IF (bEnable) THEN
	IF (bNull) THEN
		F_BACnet_MultiStatePV := E_BACnet_MultistateVal.eNull;
	ELSE
		F_BACnet_MultiStatePV := MAX(nState, E_BACnet_MultistateVal.eMin);
	END_IF
ELSE
	F_BACnet_MultiStatePV := E_BACnet_MultistateVal.eNothing;
END_IF

END_FUNCTION

// POUs/Helper/NC/F_BACnet_DeviceRecipient
// Returns an initialized recipient structure.
FUNCTION F_BACnet_DeviceRecipient : ST_BACnet_Recipient
VAR_INPUT
	nDeviceInstance		: UDINT			:= BACnet_Globals.nBACnetInstId_Auto;
END_VAR

F_BACnet_DeviceRecipient.eRecipientChoice := E_BACnet_RecipientChoice.eDevice;
F_BACnet_DeviceRecipient.stEntry.nDeviceInstance := F_BACnet_GetObjId(E_BACnetObjType.ObjDevice,nDeviceInstance);

END_FUNCTION

// POUs/Helper/NC/F_BACnet_EthernetRecipient
// Returns an initialized recipient structure.
FUNCTION F_BACnet_EthernetRecipient : ST_BACnet_Recipient
VAR_INPUT
	nIPAddress1		: BYTE;
	nIPAddress2		: BYTE;
	nIPAddress3		: BYTE;
	nIPAddress4		: BYTE;
	nPort			: UINT;
	nNetworkNr		: UINT;
END_VAR
VAR
	_nPort			: POINTER TO ARRAY[0 .. 1] OF BYTE := ADR(nPort);
END_VAR

F_BACnet_EthernetRecipient.eRecipientChoice := E_BACnet_RecipientChoice.eAddress;
F_BACnet_EthernetRecipient.stEntry.stNetAddr.eChoice := E_BACnet_AddressChoice.eEthernet;
F_BACnet_EthernetRecipient.stEntry.stNetAddr.nNetworkNr := nNetworkNr;
F_BACnet_EthernetRecipient.stEntry.stNetAddr.aAddress[0] := nIPAddress1;
F_BACnet_EthernetRecipient.stEntry.stNetAddr.aAddress[1] := nIPAddress2;
F_BACnet_EthernetRecipient.stEntry.stNetAddr.aAddress[2] := nIPAddress3;
F_BACnet_EthernetRecipient.stEntry.stNetAddr.aAddress[3] := nIPAddress4;

// Swap Port-Bytes:
F_BACnet_EthernetRecipient.stEntry.stNetAddr.aAddress[4] := _nPort^[1];
F_BACnet_EthernetRecipient.stEntry.stNetAddr.aAddress[5] := _nPort^[0];

END_FUNCTION

// POUs/Helper/NC/F_BACnet_EthernetRecipientEx
// Returns an initialized recipient structure.
FUNCTION F_BACnet_EthernetRecipientEx : ST_BACnet_Recipient
VAR_INPUT
	tIPAddress		: T_IPv4AddrArr;
	nPort			: UINT;
	nNetworkNr		: UINT;
END_VAR

F_BACnet_EthernetRecipientEx := F_BACnet_EthernetRecipient(tIPAddress[0], tIPAddress[1], tIPAddress[2], tIPAddress[3], nPort, nNetworkNr);

END_FUNCTION

// POUs/Helper/Real/F_BACnet_EnRealPV
FUNCTION F_BACnet_EnRealPV : DWORD
VAR_INPUT
	bEnable	: BOOL;
	fValue	: REAL;
END_VAR
VAR
	pDword : POINTER TO DWORD;
END_VAR

IF (bEnable) THEN
	pDword := ADR(fValue);
	F_BACnet_EnRealPV := pDword^;
ELSE
	F_BACnet_EnRealPV := F_BACnet_RealNull();
END_IF

END_FUNCTION

// POUs/Helper/Real/F_BACnet_IsFinite
FUNCTION F_BACnet_IsFinite : BOOL
VAR_INPUT
	fValue		: REAL;
END_VAR
VAR
	fArg		: T_Arg;
END_VAR

fArg.cbLen := SIZEOF(fValue);
fArg.eType := ARGTYPE_REAL;
fArg.pData := ADR(fValue);
F_BACnet_IsFinite := IsFinite(fArg);

END_FUNCTION

// POUs/Helper/Real/F_BACnet_RealEQ
FUNCTION F_BACnet_RealEQ : BOOL
VAR_INPUT
	fIn1	: REAL;
	fIn2	: REAL;
END_VAR
VAR
END_VAR

IF (F_BACnet_IsFinite(fIn1) <> F_BACnet_IsFinite(fIn2)) THEN
	F_BACnet_RealEQ := FALSE;
	RETURN;
END_IF
IF F_BACnet_IsFinite(fIn1) THEN
	IF (fIn1 <> fIn2) THEN
		F_BACnet_RealEQ := FALSE;
		RETURN;
	END_IF
END_IF
F_BACnet_RealEQ := TRUE;

END_FUNCTION

// POUs/Helper/Real/F_BACnet_RealGE
FUNCTION F_BACnet_RealGE : BOOL
VAR_INPUT
	fIn1	: REAL;
	fIn2	: REAL;
END_VAR
VAR
END_VAR

IF NOT (F_BACnet_IsFinite(fIn1) OR F_BACnet_IsFinite(fIn2)) THEN
	F_BACnet_RealGE := FALSE;
	RETURN;
END_IF
F_BACnet_RealGE := (fIn1 >= fIn2);

END_FUNCTION

// POUs/Helper/Real/F_BACnet_RealGT
FUNCTION F_BACnet_RealGT : BOOL
VAR_INPUT
	fIn1	: REAL;
	fIn2	: REAL;
END_VAR
VAR
END_VAR

IF NOT (F_BACnet_IsFinite(fIn1) OR F_BACnet_IsFinite(fIn2)) THEN
	F_BACnet_RealGT := FALSE;
	RETURN;
END_IF
F_BACnet_RealGT := (fIn1 > fIn2);

END_FUNCTION

// POUs/Helper/Real/F_BACnet_RealLE
FUNCTION F_BACnet_RealLE : BOOL
VAR_INPUT
	fIn1	: REAL;
	fIn2	: REAL;
END_VAR
VAR
END_VAR

IF NOT (F_BACnet_IsFinite(fIn1) OR F_BACnet_IsFinite(fIn2)) THEN
	F_BACnet_RealLE := FALSE;
	RETURN;
END_IF
F_BACnet_RealLE := (fIn1 <= fIn2);

END_FUNCTION

// POUs/Helper/Real/F_BACnet_RealLT
FUNCTION F_BACnet_RealLT : BOOL
VAR_INPUT
	fIn1	: REAL;
	fIn2	: REAL;
END_VAR
VAR
END_VAR

IF NOT (F_BACnet_IsFinite(fIn1) OR F_BACnet_IsFinite(fIn2)) THEN
	F_BACnet_RealLT := FALSE;
	RETURN;
END_IF
F_BACnet_RealLT := (fIn1 < fIn2);

END_FUNCTION

// POUs/Helper/Real/F_BACnet_RealNothing
FUNCTION F_BACnet_RealNothing : DWORD

F_BACnet_RealNothing:=16#7FFFFFFF;

END_FUNCTION

// POUs/Helper/Real/F_BACnet_RealPV
FUNCTION F_BACnet_RealPV : DWORD
VAR_INPUT
	bEnable	: BOOL; (* TRUE = commit to stack, FALSE = do-nothing *)
	bNull	: BOOL; (* TRUE = clear priority, FALSE = write value from input *)
	fValue	: REAL;
END_VAR
VAR
	pDword : POINTER TO DWORD;
END_VAR

IF (bEnable) THEN
	IF (bNull) THEN
		F_BACnet_RealPV := F_BACnet_RealNull();
	ELSE
		pDword := ADR(fValue);
		F_BACnet_RealPV := pDword^;
	END_IF
ELSE
	F_BACnet_RealPV := F_BACnet_RealNothing();
END_IF

END_FUNCTION

// POUs/Helper/Real/F_BACnet_RealToStr
FUNCTION F_BACnet_RealToStr : STRING
VAR_INPUT
	pValue	: POINTER TO REAL;
END_VAR
VAR
	fArg	: T_Arg;
	pDWORD	: POINTER TO DWORD;
END_VAR

IF (pValue <> 0) THEN
	fArg.cbLen := 4;
	fArg.eType := ARGTYPE_REAL;
	fArg.pData := pValue;
	pDWORD := pValue;
	IF IsFinite(fArg) THEN
		F_BACnet_RealToStr := REAL_TO_STRING(pValue^);
	ELSE
		IF (pDWORD^ = 16#7FFF0000) THEN
			F_BACnet_RealToStr := '#NULL';
		ELSIF (pDWORD^ AND 16#80000000) = 16#80000000 THEN
			F_BACnet_RealToStr := '-#QNAN';
		ELSE
			F_BACnet_RealToStr := '#QNAN';
		END_IF
	END_IF
END_IF

END_FUNCTION

// POUs/Helper/References/F_BACnet_Reference
FUNCTION F_BACnet_Reference : ST_BACnet_ObjectPropertyReference
VAR_INPUT
	iObject				: I_BACnet_Object;
	ePropertyId			: E_BACnetPropIdentifier		:= E_BACnetPropIdentifier.PropPresentValue;
END_VAR

F_BACnet_Reference.iObject := iObject;
F_BACnet_Reference.tObjectID := BACnet_Globals.nBACnetObjId_None;
F_BACnet_Reference.ePropertyId := ePropertyId;

END_FUNCTION

// POUs/Helper/References/F_BACnet_ReferenceByID
FUNCTION F_BACnet_ReferenceByID : ST_BACnet_ObjectPropertyReference
VAR_INPUT
	tObjectID			: T_BACnet_ObjectIdentifier;
	ePropertyId			: E_BACnetPropIdentifier		:= E_BACnetPropIdentifier.PropPresentValue;
END_VAR

F_BACnet_ReferenceByID.iObject := 0;
F_BACnet_ReferenceByID.tObjectID := tObjectID;
F_BACnet_ReferenceByID.ePropertyId := ePropertyId;

END_FUNCTION

// POUs/Helper/Scheduler/Calendar/F_BACnet_SchedCalendar
// Returns an initialized analog weekly scheduler.
FUNCTION F_BACnet_SchedCalendar : T_BACnet_SchedCalendar
VAR_INPUT
	iRefCalendar1	: I_BACnet_Cal	:= 0;
	iRefCalendar2	: I_BACnet_Cal	:= 0;
	iRefCalendar3	: I_BACnet_Cal	:= 0;
END_VAR
VAR
	nIndex			: INT;
END_VAR

F_BACnet_SchedCalendar[1].iRefCalendar := iRefCalendar1;

nIndex := 2;
IF (BACnet_Param.nSched_CalendarCount >= nIndex) THEN
	F_BACnet_SchedCalendar[nIndex].iRefCalendar := iRefCalendar2;
END_IF

nIndex := 3;
IF (BACnet_Param.nSched_CalendarCount >= nIndex) THEN
	F_BACnet_SchedCalendar[nIndex].iRefCalendar := iRefCalendar3;
END_IF

END_FUNCTION

// POUs/Helper/Scheduler/Exception/F_BACnet_SchedEntry1xA
// Returns an initialized analog weekly scheduler.
FUNCTION F_BACnet_SchedEntry1xA : T_BACnet_SchedExceptionEntryList
VAR_INPUT
	tEntry1Time		: TIME;
	fEntry1Value	: REAL;
END_VAR

F_BA_SetSchedulerEntry(F_BACnet_SchedEntry1xA[1], tEntry1Time, F_BA_RVal(fEntry1Value));

END_FUNCTION

// POUs/Helper/Scheduler/Exception/F_BACnet_SchedEntry1xB
// Returns an initialized binary weekly scheduler.
FUNCTION F_BACnet_SchedEntry1xB : T_BACnet_SchedExceptionEntryList
VAR_INPUT
	tEntry1Time		: TIME;
	bEntry1Value	: BOOL;
END_VAR

F_BA_SetSchedulerEntry(F_BACnet_SchedEntry1xB[1], tEntry1Time, F_BA_BVal(bEntry1Value));

END_FUNCTION

// POUs/Helper/Scheduler/Exception/F_BACnet_SchedEntry1xM
// Returns an initialized multistate weekly scheduler.
FUNCTION F_BACnet_SchedEntry1xM : T_BACnet_SchedExceptionEntryList
VAR_INPUT
	tEntry1Time		: TIME;
	nEntry1Value	: UDINT;
END_VAR

F_BA_SetSchedulerEntry(F_BACnet_SchedEntry1xM[1], tEntry1Time, F_BA_UDIVal(nEntry1Value));

END_FUNCTION

// POUs/Helper/Scheduler/Exception/F_BACnet_SchedEntry3xA
// Returns an initialized analog weekly scheduler.
FUNCTION F_BACnet_SchedEntry3xA : T_BACnet_SchedExceptionEntryList
VAR_INPUT
	tEntry1Time		: TIME;
	fEntry1Value	: REAL;
	tEntry2Time		: TIME;
	fEntry2Value	: REAL;
	tEntry3Time		: TIME;
	fEntry3Value	: REAL;
END_VAR

F_BA_SetSchedulerEntry(F_BACnet_SchedEntry3xA[1], tEntry1Time, F_BA_RVal(fEntry1Value));
F_BA_SetSchedulerEntry(F_BACnet_SchedEntry3xA[2], tEntry2Time, F_BA_RVal(fEntry2Value));
F_BA_SetSchedulerEntry(F_BACnet_SchedEntry3xA[3], tEntry3Time, F_BA_RVal(fEntry3Value));

END_FUNCTION

// POUs/Helper/Scheduler/Exception/F_BACnet_SchedEntry3xB
// Returns an initialized binary weekly scheduler.
FUNCTION F_BACnet_SchedEntry3xB : T_BACnet_SchedExceptionEntryList
VAR_INPUT
	tEntry1Time		: TIME;
	bEntry1Value	: BOOL;
	tEntry2Time		: TIME;
	bEntry2Value	: BOOL;
	tEntry3Time		: TIME;
	bEntry3Value	: BOOL;
END_VAR

F_BA_SetSchedulerEntry(F_BACnet_SchedEntry3xB[1], tEntry1Time, F_BA_BVal(bEntry1Value));
F_BA_SetSchedulerEntry(F_BACnet_SchedEntry3xB[2], tEntry2Time, F_BA_BVal(bEntry2Value));
F_BA_SetSchedulerEntry(F_BACnet_SchedEntry3xB[3], tEntry3Time, F_BA_BVal(bEntry3Value));

END_FUNCTION

// POUs/Helper/Scheduler/Exception/F_BACnet_SchedEntry3xM
// Returns an initialized multistate weekly scheduler.
FUNCTION F_BACnet_SchedEntry3xM : T_BACnet_SchedExceptionEntryList
VAR_INPUT
	tEntry1Time		: TIME;
	nEntry1Value	: UDINT;
	tEntry2Time		: TIME;
	nEntry2Value	: UDINT;
	tEntry3Time		: TIME;
	nEntry3Value	: UDINT;
END_VAR

F_BA_SetSchedulerEntry(F_BACnet_SchedEntry3xM[1], tEntry1Time, F_BA_UDIVal(nEntry1Value));
F_BA_SetSchedulerEntry(F_BACnet_SchedEntry3xM[2], tEntry2Time, F_BA_UDIVal(nEntry2Value));
F_BA_SetSchedulerEntry(F_BACnet_SchedEntry3xM[3], tEntry3Time, F_BA_UDIVal(nEntry3Value));

END_FUNCTION

// POUs/Helper/Scheduler/Exception/F_BACnet_SchedEntry5xA
// Returns an initialized analog weekly scheduler.
FUNCTION F_BACnet_SchedEntry5xA : T_BACnet_SchedExceptionEntryList
VAR_INPUT
	tEntry1Time		: TIME;
	fEntry1Value	: REAL;
	tEntry2Time		: TIME;
	fEntry2Value	: REAL;
	tEntry3Time		: TIME;
	fEntry3Value	: REAL;
	tEntry4Time		: TIME;
	fEntry4Value	: REAL;
	tEntry5Time		: TIME;
	fEntry5Value	: REAL;
END_VAR

F_BA_SetSchedulerEntry(F_BACnet_SchedEntry5xA[1], tEntry1Time, F_BA_RVal(fEntry1Value));
F_BA_SetSchedulerEntry(F_BACnet_SchedEntry5xA[2], tEntry2Time, F_BA_RVal(fEntry2Value));
F_BA_SetSchedulerEntry(F_BACnet_SchedEntry5xA[3], tEntry3Time, F_BA_RVal(fEntry3Value));
F_BA_SetSchedulerEntry(F_BACnet_SchedEntry5xA[4], tEntry4Time, F_BA_RVal(fEntry4Value));
F_BA_SetSchedulerEntry(F_BACnet_SchedEntry5xA[5], tEntry5Time, F_BA_RVal(fEntry5Value));

END_FUNCTION

// POUs/Helper/Scheduler/Exception/F_BACnet_SchedEntry5xB
// Returns an initialized binary weekly scheduler.
FUNCTION F_BACnet_SchedEntry5xB : T_BACnet_SchedExceptionEntryList
VAR_INPUT
	tEntry1Time		: TIME;
	bEntry1Value	: BOOL;
	tEntry2Time		: TIME;
	bEntry2Value	: BOOL;
	tEntry3Time		: TIME;
	bEntry3Value	: BOOL;
	tEntry4Time		: TIME;
	bEntry4Value	: BOOL;
	tEntry5Time		: TIME;
	bEntry5Value	: BOOL;
END_VAR

F_BA_SetSchedulerEntry(F_BACnet_SchedEntry5xB[1], tEntry1Time, F_BA_BVal(bEntry1Value));
F_BA_SetSchedulerEntry(F_BACnet_SchedEntry5xB[2], tEntry2Time, F_BA_BVal(bEntry2Value));
F_BA_SetSchedulerEntry(F_BACnet_SchedEntry5xB[3], tEntry3Time, F_BA_BVal(bEntry3Value));
F_BA_SetSchedulerEntry(F_BACnet_SchedEntry5xB[4], tEntry4Time, F_BA_BVal(bEntry4Value));
F_BA_SetSchedulerEntry(F_BACnet_SchedEntry5xB[5], tEntry5Time, F_BA_BVal(bEntry5Value));

END_FUNCTION

// POUs/Helper/Scheduler/Exception/F_BACnet_SchedEntry5xM
// Returns an initialized multistate weekly scheduler.
FUNCTION F_BACnet_SchedEntry5xM : T_BACnet_SchedExceptionEntryList
VAR_INPUT
	tEntry1Time		: TIME;
	nEntry1Value	: UDINT;
	tEntry2Time		: TIME;
	nEntry2Value	: UDINT;
	tEntry3Time		: TIME;
	nEntry3Value	: UDINT;
	tEntry4Time		: TIME;
	nEntry4Value	: UDINT;
	tEntry5Time		: TIME;
	nEntry5Value	: UDINT;
END_VAR

F_BA_SetSchedulerEntry(F_BACnet_SchedEntry5xM[1], tEntry1Time, F_BA_UDIVal(nEntry1Value));
F_BA_SetSchedulerEntry(F_BACnet_SchedEntry5xM[2], tEntry2Time, F_BA_UDIVal(nEntry2Value));
F_BA_SetSchedulerEntry(F_BACnet_SchedEntry5xM[3], tEntry3Time, F_BA_UDIVal(nEntry3Value));
F_BA_SetSchedulerEntry(F_BACnet_SchedEntry5xM[4], tEntry4Time, F_BA_UDIVal(nEntry4Value));
F_BA_SetSchedulerEntry(F_BACnet_SchedEntry5xM[5], tEntry5Time, F_BA_UDIVal(nEntry5Value));

END_FUNCTION

// POUs/Helper/Scheduler/Weekly/F_BACnet_SchedWeekly3xA
// Returns an initialized analog weekly scheduler.
FUNCTION F_BACnet_SchedWeekly3xA : T_BACnet_SchedWeek
VAR_INPUT
	eDayFrom		: E_BA_Weekday		:= E_BA_Weekday.eMonday;
	eDayTo			: E_BA_Weekday		:= E_BA_Weekday.eSunday;
	
	tEntry1Time		: TIME;
	fEntry1Value	: REAL;
	tEntry2Time		: TIME;
	fEntry2Value	: REAL;
	tEntry3Time		: TIME;
	fEntry3Value	: REAL;
END_VAR

F_BA_SetWeekdays(F_BACnet_SchedWeekly3xA, eDayFrom, eDayTo, 1, tEntry1Time, F_BA_RVal(fEntry1Value));
F_BA_SetWeekdays(F_BACnet_SchedWeekly3xA, eDayFrom, eDayTo, 2, tEntry2Time, F_BA_RVal(fEntry2Value));
F_BA_SetWeekdays(F_BACnet_SchedWeekly3xA, eDayFrom, eDayTo, 3, tEntry3Time, F_BA_RVal(fEntry3Value));

END_FUNCTION

// POUs/Helper/Scheduler/Weekly/F_BACnet_SchedWeekly3xB
// Returns an initialized binary weekly scheduler.
FUNCTION F_BACnet_SchedWeekly3xB : T_BACnet_SchedWeek
VAR_INPUT
	eDayFrom		: E_BA_Weekday		:= E_BA_Weekday.eMonday;
	eDayTo			: E_BA_Weekday		:= E_BA_Weekday.eSunday;
	
	tEntry1Time		: TIME;
	bEntry1Value	: BOOL;
	tEntry2Time		: TIME;
	bEntry2Value	: BOOL;
	tEntry3Time		: TIME;
	bEntry3Value	: BOOL;
END_VAR

F_BA_SetWeekdays(F_BACnet_SchedWeekly3xB, eDayFrom, eDayTo, 1, tEntry1Time, F_BA_BVal(bEntry1Value));
F_BA_SetWeekdays(F_BACnet_SchedWeekly3xB, eDayFrom, eDayTo, 2, tEntry2Time, F_BA_BVal(bEntry2Value));
F_BA_SetWeekdays(F_BACnet_SchedWeekly3xB, eDayFrom, eDayTo, 3, tEntry3Time, F_BA_BVal(bEntry3Value));

END_FUNCTION

// POUs/Helper/Scheduler/Weekly/F_BACnet_SchedWeekly3xM
// Returns an initialized multistate weekly scheduler.
FUNCTION F_BACnet_SchedWeekly3xM : T_BACnet_SchedWeek
VAR_INPUT
	eDayFrom		: E_BA_Weekday		:= E_BA_Weekday.eMonday;
	eDayTo			: E_BA_Weekday		:= E_BA_Weekday.eSunday;
	
	tEntry1Time		: TIME;
	nEntry1Value	: UDINT;
	tEntry2Time		: TIME;
	nEntry2Value	: UDINT;
	tEntry3Time		: TIME;
	nEntry3Value	: UDINT;
END_VAR

F_BA_SetWeekdays(F_BACnet_SchedWeekly3xM, eDayFrom, eDayTo, 1, tEntry1Time, F_BA_UDIVal(nEntry1Value));
F_BA_SetWeekdays(F_BACnet_SchedWeekly3xM, eDayFrom, eDayTo, 2, tEntry2Time, F_BA_UDIVal(nEntry2Value));
F_BA_SetWeekdays(F_BACnet_SchedWeekly3xM, eDayFrom, eDayTo, 3, tEntry3Time, F_BA_UDIVal(nEntry3Value));

END_FUNCTION

// POUs/Helper/Scheduler/Weekly/F_BACnet_SchedWeekly5xA
// Returns an initialized analog weekly scheduler.
FUNCTION F_BACnet_SchedWeekly5xA : T_BACnet_SchedWeek
VAR_INPUT
	eDayFrom		: E_BA_Weekday		:= E_BA_Weekday.eMonday;
	eDayTo			: E_BA_Weekday		:= E_BA_Weekday.eSunday;
	
	tEntry1Time		: TIME;
	fEntry1Value	: REAL;
	tEntry2Time		: TIME;
	fEntry2Value	: REAL;
	tEntry3Time		: TIME;
	fEntry3Value	: REAL;
	tEntry4Time		: TIME;
	fEntry4Value	: REAL;
	tEntry5Time		: TIME;
	fEntry5Value	: REAL;
END_VAR

F_BA_SetWeekdays(F_BACnet_SchedWeekly5xA, eDayFrom, eDayTo, 1, tEntry1Time, F_BA_RVal(fEntry1Value));
F_BA_SetWeekdays(F_BACnet_SchedWeekly5xA, eDayFrom, eDayTo, 2, tEntry2Time, F_BA_RVal(fEntry2Value));
F_BA_SetWeekdays(F_BACnet_SchedWeekly5xA, eDayFrom, eDayTo, 3, tEntry3Time, F_BA_RVal(fEntry3Value));
F_BA_SetWeekdays(F_BACnet_SchedWeekly5xA, eDayFrom, eDayTo, 4, tEntry4Time, F_BA_RVal(fEntry4Value));
F_BA_SetWeekdays(F_BACnet_SchedWeekly5xA, eDayFrom, eDayTo, 5, tEntry5Time, F_BA_RVal(fEntry5Value));

END_FUNCTION

// POUs/Helper/Scheduler/Weekly/F_BACnet_SchedWeekly5xB
// Returns an initialized binary weekly scheduler.
FUNCTION F_BACnet_SchedWeekly5xB : T_BACnet_SchedWeek
VAR_INPUT
	eDayFrom		: E_BA_Weekday		:= E_BA_Weekday.eMonday;
	eDayTo			: E_BA_Weekday		:= E_BA_Weekday.eSunday;
	
	tEntry1Time		: TIME;
	bEntry1Value	: BOOL;
	tEntry2Time		: TIME;
	bEntry2Value	: BOOL;
	tEntry3Time		: TIME;
	bEntry3Value	: BOOL;
	tEntry4Time		: TIME;
	bEntry4Value	: BOOL;
	tEntry5Time		: TIME;
	bEntry5Value	: BOOL;
END_VAR

F_BA_SetWeekdays(F_BACnet_SchedWeekly5xB, eDayFrom, eDayTo, 1, tEntry1Time, F_BA_BVal(bEntry1Value));
F_BA_SetWeekdays(F_BACnet_SchedWeekly5xB, eDayFrom, eDayTo, 2, tEntry2Time, F_BA_BVal(bEntry2Value));
F_BA_SetWeekdays(F_BACnet_SchedWeekly5xB, eDayFrom, eDayTo, 3, tEntry3Time, F_BA_BVal(bEntry3Value));
F_BA_SetWeekdays(F_BACnet_SchedWeekly5xB, eDayFrom, eDayTo, 4, tEntry4Time, F_BA_BVal(bEntry4Value));
F_BA_SetWeekdays(F_BACnet_SchedWeekly5xB, eDayFrom, eDayTo, 5, tEntry5Time, F_BA_BVal(bEntry5Value));

END_FUNCTION

// POUs/Helper/Scheduler/Weekly/F_BACnet_SchedWeekly5xM
// Returns an initialized multistate weekly scheduler.
FUNCTION F_BACnet_SchedWeekly5xM : T_BACnet_SchedWeek
VAR_INPUT
	eDayFrom		: E_BA_Weekday		:= E_BA_Weekday.eMonday;
	eDayTo			: E_BA_Weekday		:= E_BA_Weekday.eSunday;
	
	tEntry1Time		: TIME;
	nEntry1Value	: UDINT;
	tEntry2Time		: TIME;
	nEntry2Value	: UDINT;
	tEntry3Time		: TIME;
	nEntry3Value	: UDINT;
	tEntry4Time		: TIME;
	nEntry4Value	: UDINT;
	tEntry5Time		: TIME;
	nEntry5Value	: UDINT;
END_VAR

F_BA_SetWeekdays(F_BACnet_SchedWeekly5xM, eDayFrom, eDayTo, 1, tEntry1Time, F_BA_UDIVal(nEntry1Value));
F_BA_SetWeekdays(F_BACnet_SchedWeekly5xM, eDayFrom, eDayTo, 2, tEntry2Time, F_BA_UDIVal(nEntry2Value));
F_BA_SetWeekdays(F_BACnet_SchedWeekly5xM, eDayFrom, eDayTo, 3, tEntry3Time, F_BA_UDIVal(nEntry3Value));
F_BA_SetWeekdays(F_BACnet_SchedWeekly5xM, eDayFrom, eDayTo, 4, tEntry4Time, F_BA_UDIVal(nEntry4Value));
F_BA_SetWeekdays(F_BACnet_SchedWeekly5xM, eDayFrom, eDayTo, 5, tEntry5Time, F_BA_UDIVal(nEntry5Value));

END_FUNCTION

// POUs/Helper/String/F_BACnet_GetObjectIdString
FUNCTION F_BACnet_GetObjectIdString : STRING
VAR_INPUT
	tObjectID : T_BACnet_ObjectIdentifier := 16#FFFFFFFF;
END_VAR
VAR
	nObjType	: DINT;
	nObjInstance: UDINT;
END_VAR

nObjType	:= F_BACnet_GetObjType(tObjectID);
nObjInstance:= F_BACnet_GetObjInstance(tObjectID);
IF (BACnet_Globals.nRange_ObjectTypeFirst <= nObjType) AND (nObjType <= BACnet_Globals.nRange_ObjectTypeLast) THEN
	F_BACnet_GetObjectIdString := CONCAT(CONCAT(BACnet_Globals.aSpec_ObjectTypeShortcut[nObjType], ':'), UDINT_TO_STRING(nObjInstance));
ELSE
	F_BACnet_GetObjectIdString := CONCAT('???:', UDINT_TO_STRING(nObjInstance));
END_IF

END_FUNCTION

// POUs/Helper/String/FB_BACnet_StringExtEncode
FUNCTION_BLOCK FB_BACnet_StringExtEncode (* convert Windows-1252 to ANSI/UTF-8 BACnet Character String *)
VAR_INPUT
	pString			: POINTER TO T_MaxString; (* pointer to Windows-1252 encoded PLC text *)
	nSize			: INT; (* string length or data size of pText field *)
	pResultExtStr	: POINTER TO ST_BACnet_CharacterStringExt;
	nResult		: UDINT; (* byte size of result data field *)
END_VAR
VAR_OUTPUT
	bValid			: BOOL;
	bOverflow		: BOOL; (* String length overflow (source string too long) *)
	nLength			: UDINT; (* out string data length in byte *)
END_VAR

(* preset valid to FALSE *)
bOverflow := FALSE;
bValid := TRUE;
(* check pointer *)
IF (pString = 0) OR (pResultExtStr = 0) THEN
	nLength := 0;
	bValid := FALSE;
	RETURN;
END_IF

(* clear string *)
MEMSET(destAddr:=pResultExtStr, fillByte:=0, n:=nResult);
(* check input size *)
IF (nSize <= 0) THEN
	nLength := 0;

(* convert *)
ELSE
	IF (F_BACnet_EncodeUTF8(
		pString		:= pString,
		nString	:= TO_UDINT(nSize),
		pResult		:= pResultExtStr,
		nResult	:= nResult,
		nResultLen	:= nLength) > nResult)
	THEN
		bOverflow	:= TRUE;
		bValid		:= FALSE;
	END_IF
END_IF

END_FUNCTION_BLOCK

// POUs/Helper/F_BACnet_GetObjectListIndex
FUNCTION F_BACnet_GetObjectListIndex : DINT
VAR_INPUT
	tObjectId	: T_BACnet_ObjectIdentifier := 16#FFFFFFFF;
END_VAR

VAR
	nMax : DINT;
	i : DINT;
END_VAR
(*All VAR_IN_OUT variables have been moved to the end of the declaration due to compatibility reasons*)
VAR_IN_OUT
	stObjIDList	: ST_BACnet_ObjectIdentifierList;
END_VAR

nMax := UDINT_TO_DINT(stObjIDList.nEntries)-1;
F_BACnet_GetObjectListIndex := -1; (* preset: no match *)
FOR i := 0 TO nMax DO
	IF stObjIDList.aObjList[i] = tObjectId THEN
		F_BACnet_GetObjectListIndex := i; (* match *)
		RETURN;
	END_IF
END_FOR

END_FUNCTION

// POUs/Helper/FB_BACnet_AvgValue
FUNCTION_BLOCK FB_BACnet_AvgValue
VAR_INPUT
	X	: REAL; (* input value to average *)
	n	: UINT; (* number of averages (0 = no average --> Y = X) *)
END_VAR
VAR_OUTPUT
	Y	: REAL; (* average result *)
END_VAR
VAR
	_n	: UINT := 0;
	_Xn : LREAL;
END_VAR

IF (_n > n) THEN
	_n := n;
END_IF
IF (_n = 0) OR (n = 0) THEN
	_Xn := REAL_TO_LREAL(X);
ELSE
	_Xn := ((_Xn * _n) + REAL_TO_LREAL(X)) / UINT_TO_LREAL(_n + 1);
END_IF
_n := _n + 1;
Y := LREAL_TO_REAL(_Xn);

END_FUNCTION_BLOCK

// POUs/Local/Objects/[Base]/FB_BACnet_BaseTLog
FUNCTION_BLOCK FB_BACnet_BaseTLog EXTENDS FB_BACnet_EventObject
VAR_INPUT CONSTANT PERSISTENT
	{region 'Fixed Parameters'}
		{attribute 'parameterCategory':='Value'}
		nBufferSize : UDINT := BACnet_Param.nTLog_ArraySize;
	{endregion}
	{region 'Variable Parameters'}
		{attribute 'parameterCategory':='State'}
		bLogEnable : BOOL;
		
		{attribute 'parameterCategory':='Config'}
		stStartTime : ST_BA_DateTime;
		{attribute 'parameterCategory':='Config'}
		stStopTime : ST_BA_DateTime;
		{attribute 'parameterCategory':='Config'}
		bStopWhenFull : BOOL;
		{attribute 'parameterCategory':='Config'}
		{attribute 'parameterUnit':= '1/100s'}
		nLogInterval : UDINT := 90000;
		{attribute 'parameterCategory':='Config'}
		nNotificationThreshold : UDINT := 50;
		{attribute 'parameterCategory':='Config'}
		eLoggingType : E_BA_LoggingType := E_BA_LoggingType.ePolled;
	{endregion}
END_VAR
VAR_OUTPUT
	nRecordCount				: UDINT;
	nTotalRecordCount			: UDINT;
END_VAR

SUPER^();

METHOD PROTECTED OnObjectStateChanged
VAR
	_pBufferVal		: PVOID;
	_nBufferSize	: DINT;
END_VAR
SUPER^.OnObjectStateChanged();

CASE (tState) OF
	TCOM_STATE.TCOM_STATE_PREOP:
		// SyncHandler:
		RequestSyncHandlers(2, 7);
		
		// Properties:
		// May limit buffer size to respect array size:
		nBufferSize := MIN(BACnet_Param.nTLog_ArraySize, nBufferSize);
		
		WritePropertyUDInt(E_BACnetPropIdentifier.PropBufferSize, nBufferSize);
		
	TCOM_STATE.TCOM_STATE_SAFEOP:
		;

	TCOM_STATE.TCOM_STATE_OP:
		// Synchronize:
		SyncProperty(E_BACnetPropIdentifier.PropRecordCount, SIZEOF(nRecordCount), ADR(nRecordCount), 0, eSync_FromSupplement, FALSE);
		SyncProperty(E_BACnetPropIdentifier.PropTotalRecordCount, SIZEOF(nTotalRecordCount), ADR(nTotalRecordCount), 0, eSync_FromSupplement, FALSE);
		
		SyncProperty(E_BACnetPropIdentifier.PropEnable, SIZEOF(bLogEnable), ADR(bLogEnable), 0, eFullSync_InitPLC, FALSE);
		SyncProperty(E_BACnetPropIdentifier.PropStartTime, SIZEOF(stStartTime), ADR(stStartTime), 0, eFullSync_InitPLC, FALSE);
		SyncProperty(E_BACnetPropIdentifier.PropStopTime, SIZEOF(stStopTime), ADR(stStopTime), 0, eFullSync_InitPLC, FALSE);
		SyncProperty(E_BACnetPropIdentifier.PropStopWhenFull, SIZEOF(bStopWhenFull), ADR(bStopWhenFull), 0, eFullSync_InitPLC, FALSE);
		SyncProperty(E_BACnetPropIdentifier.PropLogInterval, SIZEOF(nLogInterval), ADR(nLogInterval), 0, eFullSync_InitPLC, FALSE);
		SyncProperty(E_BACnetPropIdentifier.PropNotificationThreshold, SIZEOF(nNotificationThreshold), ADR(nNotificationThreshold), 0, eFullSync_InitPLC, FALSE);
		SyncProperty(E_BACnetPropIdentifier.PropLoggingType, SIZEOF(eLoggingType), ADR(eLoggingType), 0, eFullSync_InitPLC, FALSE);
		
END_CASE
END_METHOD

END_FUNCTION_BLOCK

// POUs/Local/Objects/[Internal]/Property/Buffer/[Archiv]/FB_BACnet_WeeklyScheduleBuffer
FUNCTION_BLOCK INTERNAL FB_BACnet_WeeklyScheduleBuffer EXTENDS FB_BACnet_BaseListBuffer

SUPER^();

METHOD FB_init : BOOL
VAR_INPUT
	bInitRetains : BOOL; // if TRUE, the retain variables are initialized (warm start / cold start)
	bInCopyCode : BOOL;  // if TRUE, the instance afterwards gets moved into the copy code (online change)
END_VAR
ePropertyID := E_BACnetPropIdentifier.PropWeeklySchedule;
END_METHOD

METHOD ResetValue
VAR
	_nDay : INT;
END_VAR
SUPER^.ResetValue();

// Write empty weekday-array to buffer:
FOR _nDay := E_BA_Weekday.First TO E_BA_Weekday.Last DO
	MemSetULINT(16#0000000080000008, nUsedSize);
	MemSetULINT(16#0000000000000000, nUsedSize);
END_FOR

(*
FOR iDayTmp := iWeekdayFirst TO iWeekdayLast DO
	MemSetULINT(16#0000000080000020, nUsedSize);
	MemSetULINT(16#0000000000000000, nUsedSize);
	MemSetULINT(16#0000000000000000, nUsedSize);
	MemSetULINT(16#0000000000000000, nUsedSize);
	MemSetULINT(16#0000000000000000, nUsedSize);
END_FOR
*)
END_METHOD

END_FUNCTION_BLOCK

// POUs/Local/Objects/[Internal]/Property/Buffer/Base/FB_BACnet_BaseListBuffer
FUNCTION_BLOCK INTERNAL FB_BACnet_BaseListBuffer EXTENDS FB_BACnet_BasePropertyBuffer
VAR PERSISTENT
	aBuffer : ARRAY[1 .. nBACnet_BufferSize] OF BYTE;
END_VAR
VAR CONSTANT
	{attribute 'hide'}
	{attribute 'parameterUnit':= 'byte'}
	nBACnet_BufferSize	: UINT	:= 8192;
END_VAR

SUPER^();

METHOD PROTECTED ValidateInst : BOOL
nBufferSize := SIZEOF(aBuffer);
pBufferValue := ADR(aBuffer);

ValidateInst := SUPER^.ValidateInst();
END_METHOD

END_FUNCTION_BLOCK

// POUs/Local/Objects/[Internal]/Property/Buffer/Base/FB_BACnet_BasePropertyBuffer
FUNCTION_BLOCK INTERNAL FB_BACnet_BasePropertyBuffer
VAR_OUTPUT
	ePropertyID : E_BACnetPropIdentifier := E_BACnetPropIdentifier.PropInvalid;		// ID of referred property
	bChangeTrig : BOOL;												// Change trigger
	nChanges : UINT;												// Changes counter
	bReady : BOOL;												// Synchronization of referred property successfully initialized
END_VAR
VAR PERSISTENT
	nUsedSize : UDINT;
END_VAR
VAR
	// Init via instance-declaration:
	iRefObject : I_BACnet_Object;
	
	// Init via SubClass:
	tSyncState : TCOM_STATE := TCOM_STATE.TCOM_STATE_OP;						// Object-state to init synchronization of referred property
END_VAR
VAR_STAT
	// (BETA) ... Following symbols should be made non-static / thread safe!
	// Use "ValidateInst()" to ensure data to be valid: 
	fbRefObject : POINTER TO FB_BACnet_Object;
	nBufferSize : UDINT;
	pBufferValue : PVOID;
END_VAR
(*
VAR
	// [DEBUG]:
	eDebugCommand : (eNone:=1, eReadBuffer:=2, eWriteBuffer:=3, eResetBuffer:=4, ePrintBuffer:=5) UDINT := 1;
	sDebugHexBuffer : T_MaxString;
END_VAR
*)

IF (bChangeTrig) THEN
	bChangeTrig := FALSE;
	nChanges := (nChanges+1);
	
	IF (ValidateInst()) THEN
		// Refresh property value:
		ReadValue();
	END_IF
END_IF

(*
// [DEBUG]:
IF (eDebugCommand <> eNone) THEN
	IF (ValidateInst()) THEN
		CASE (eDebugCommand) OF
			eReadBuffer:
				ReadValue();
			eWriteBuffer:
				WriteValue();
			eResetBuffer:
				ResetValue();
			ePrintBuffer:
				sDebugHexBuffer := DATA_TO_HEXSTR(pData:=pBufferValue, cbData:=TO_UDINT(nUsedSize), FALSE);
		END_CASE
	END_IF
	eDebugCommand := eNone;
END_IF
*)

// Write a (any type) value to the memory buffer. 
// > Ensure to point to valid memory buffer via "ValidateInst()"!
METHOD PROTECTED MemSet : BOOL
VAR_INPUT
	xValue : ANY;
END_VAR
VAR_IN_OUT
	nOffset : UDINT;
END_VAR
VAR
	_nSizeTmp : UDINT;
END_VAR
_nSizeTmp := TO_UDINT(xValue.diSize);

IF (pBufferValue = 0) THEN
	F_BA_LogMessage(ADSLOG_MSGTYPE_ERROR, 'MS02', 'PropertyBuffer.MemSet: Uninitialized buffer!');
ELSIF ((_nSizeTmp+nOffset) > nBufferSize) THEN
	F_BA_LogMessage(ADSLOG_MSGTYPE_ERROR, 'MS04', 'PropertyBuffer.MemSet: Buffer size exceeded!');
ELSE
	MEMCPY((pBufferValue+nOffset), xValue.pValue, _nSizeTmp);
	nOffset := (nOffset+_nSizeTmp);
	
	MemSet := TRUE;
END_IF
END_METHOD

// Write a 1Byte-value to the memory buffer. 
METHOD PROTECTED MemSetBYTE : BOOL
VAR_INPUT
	nValue : BYTE;
END_VAR
VAR_IN_OUT
	nOffset : UDINT;
END_VAR
MemSetBYTE := MemSet(nValue, nOffset);
END_METHOD

// Write a 4Byte-value to the memory buffer. 
METHOD PROTECTED MemSetUDINT : BOOL
VAR_INPUT
	nValue : UDINT;
END_VAR
VAR_IN_OUT
	nOffset : UDINT;
END_VAR
MemSetUDINT := MemSet(nValue, nOffset);
END_METHOD

// Write a 2Byte-value to the memory buffer. 
METHOD PROTECTED MemSetUINT : BOOL
VAR_INPUT
	nValue : UINT;
END_VAR
VAR_IN_OUT
	nOffset : UDINT;
END_VAR
MemSetUINT := MemSet(nValue, nOffset);
END_METHOD

// Write a 8Byte-value to the memory buffer. 
METHOD PROTECTED MemSetULINT : BOOL
VAR_INPUT
	nValue : ULINT;
END_VAR
VAR_IN_OUT
	nOffset : UDINT;
END_VAR
MemSetULINT := MemSet(nValue, nOffset);
END_METHOD

METHOD PROTECTED ReadValue : HRESULT
nUsedSize := nBufferSize;
ReadValue := fbRefObject^.ReadProperty(ePropertyID, pBufferValue, ADR(nUsedSize));
END_METHOD

METHOD PROTECTED ValidateInst : BOOL
IF (iRefObject = 0) THEN
	F_BA_LogMessage(ADSLOG_MSGTYPE_ERROR, 'GB3', 'PropertyBuffer: Unreferred object!');
	
ELSIF (NOT __QUERYPOINTER(iRefObject, fbRefObject)) OR (fbRefObject = 0) THEN
	F_BA_LogMessage(ADSLOG_MSGTYPE_ERROR, 'GB6', 'PropertyBuffer: Invalid referred object!');
	
ELSIF (nBufferSize = 0) OR (pBufferValue = 0) THEN
	F_BA_LogMessage1(ADSLOG_MSGTYPE_ERROR, 'GB8', 'PropertyBuffer: Unimplemented buffer of property "%d"!', F_INT(ePropertyID));

ELSE
	ValidateInst := TRUE;
END_IF
END_METHOD

METHOD PROTECTED WriteValue : HRESULT
WriteValue := fbRefObject^.WriteProperty(ePropertyID, pBufferValue, TO_DINT(nUsedSize));
END_METHOD

METHOD OnObjectStateChanged
VAR_INPUT
	tState : TCOM_STATE;
END_VAR
VAR
	eSyncMode : E_BA_FullSyncMode := eFullSync_InitPLC;
END_VAR
IF (tState = tSyncState) THEN
	IF (ePropertyID = E_BACnetPropIdentifier.PropInvalid) THEN
		F_BA_LogMessage(ADSLOG_MSGTYPE_ERROR, 'OOSC3', 'PropertyBuffer: Uninitialized property type!');
		
	ELSIF (ValidateInst()) THEN
		// Initialize COV-Trigger:
		IF (fbRefObject^.SyncPropertyCOV(ePropertyID, ADR(bChangeTrig))) THEN
			// Initialize property:
			IF (nUsedSize = 0) THEN
				// Initial value has defenitly to be read from stack:
				bReady := SUCCEEDED(ReadValue());
			ELSE
				CASE (eSyncMode) OF
					eSync_ToSupplement,
					eFullSync_InitPLC:
						bReady := SUCCEEDED(WriteValue());
				ELSE
					bReady := SUCCEEDED(ReadValue());
				END_CASE
			END_IF
		END_IF
	END_IF
END_IF
END_METHOD

METHOD ResetValue
nUsedSize := 0;

ValidateInst();
END_METHOD

END_FUNCTION_BLOCK

// POUs/Local/Objects/[Internal]/Property/Buffer/Base/FB_BACnet_BaseArrayBuffer
FUNCTION_BLOCK INTERNAL FB_BACnet_BaseArrayBuffer EXTENDS FB_BACnet_BasePropertyBuffer
VAR CONSTANT
	{attribute 'hide'}
	nBACnet_EntryCount	: UINT	:= 256;
	
	// Hint:
	// > [BufferSize] := (nBACnet_EntryCount * [EntrySize])
END_VAR

SUPER^();

END_FUNCTION_BLOCK

// POUs/Local/Objects/[Internal]/Property/Buffer/Base/FB_BACnet_BasePropertyLogBuffer
FUNCTION_BLOCK FB_BACnet_BasePropertyLogBuffer EXTENDS FB_BACnet_BasePropertyBuffer

SUPER^();

METHOD OnObjectStateChanged
VAR_INPUT
	tState : TCOM_STATE;
END_VAR
VAR
	eSyncMode : E_BA_FullSyncMode := eFullSync_InitPLC;
END_VAR
IF (tState = tSyncState) THEN
	IF (ePropertyID = E_BACnetPropIdentifier.PropInvalid) THEN
		F_BA_LogMessage(ADSLOG_MSGTYPE_ERROR, 'OOSC8', 'PropertyBuffer: Uninitialized property type!');
		
	ELSIF (ValidateInst()) THEN
		// Initialize COV-Trigger:
		IF (fbRefObject^.SyncPropertyCOV(ePropertyID, ADR(bChangeTrig))) THEN
			// Initialize property:
			IF (nUsedSize = 0) THEN
				IF fbRefObject^.bIsReused THEN
					// Reset stack value:
					bReady := SUCCEEDED(fbRefObject^.WritePropertyUDInt(E_BACnetPropIdentifier.PropTotalRecordCount,0));
				ELSE
					// Initial value has defenitly to be read from stack:
					bReady := SUCCEEDED(ReadValue());
				END_IF
			ELSE
				IF fbRefObject^.bIsReused THEN
					bReady := SUCCEEDED(ReadValue());
				ELSE
					bReady := SUCCEEDED(WriteValue());
				END_IF
			END_IF
		END_IF
	END_IF
END_IF
END_METHOD

END_FUNCTION_BLOCK

// POUs/Local/Objects/[Internal]/Property/Buffer/FB_BACnet_DateListBuffer
FUNCTION_BLOCK INTERNAL FB_BACnet_DateListBuffer EXTENDS FB_BACnet_BaseListBuffer

SUPER^();

METHOD FB_init : BOOL
VAR_INPUT
	bInitRetains : BOOL; // if TRUE, the retain variables are initialized (warm start / cold start)
	bInCopyCode : BOOL;  // if TRUE, the instance afterwards gets moved into the copy code (online change)
END_VAR
ePropertyID := E_BACnetPropIdentifier.PropDateList;
END_METHOD

END_FUNCTION_BLOCK

// POUs/Local/Objects/[Internal]/Property/Buffer/FB_BACnet_EventLogBuffer
FUNCTION_BLOCK INTERNAL FB_BACnet_EventLogBuffer EXTENDS FB_BACnet_BasePropertyBuffer
VAR PERSISTENT
	aBuffer : ARRAY[1 .. nBACnet_BufferSize] OF BYTE;
END_VAR
VAR CONSTANT
	{attribute 'hide'}
	{attribute 'parameterUnit':= 'byte'}
	nBACnet_EntrySize	: UINT	:= 376;
	{attribute 'hide'}
	nBACnet_EntryCount	: UINT	:= BACnet_Globals.nDataField_MaxEventLogBufferEntries;
	
	{attribute 'hide'}
	nBACnet_BufferSize	: UINT	:= (nBACnet_EntrySize * nBACnet_EntryCount);
END_VAR

SUPER^();

METHOD PROTECTED ValidateInst : BOOL
nBufferSize := SIZEOF(aBuffer);
pBufferValue := ADR(aBuffer);

ValidateInst := SUPER^.ValidateInst();
END_METHOD

METHOD FB_init : BOOL
VAR_INPUT
	bInitRetains : BOOL; // if TRUE, the retain variables are initialized (warm start / cold start)
	bInCopyCode : BOOL;  // if TRUE, the instance afterwards gets moved into the copy code (online change)
END_VAR
ePropertyID := E_BACnetPropIdentifier.PropLogBuffer;
END_METHOD

END_FUNCTION_BLOCK

// POUs/Local/Objects/[Internal]/Property/Buffer/FB_BACnet_ExceptionScheduleBuffer
FUNCTION_BLOCK INTERNAL FB_BACnet_ExceptionScheduleBuffer EXTENDS FB_BACnet_BaseListBuffer

SUPER^();

METHOD FB_init : BOOL
VAR_INPUT
	bInitRetains : BOOL; // if TRUE, the retain variables are initialized (warm start / cold start)
	bInCopyCode : BOOL;  // if TRUE, the instance afterwards gets moved into the copy code (online change)
END_VAR
ePropertyID := E_BACnetPropIdentifier.PropExceptionSchedule;
END_METHOD

END_FUNCTION_BLOCK

// POUs/Local/Objects/[Internal]/Property/Buffer/FB_BACnet_TLMBuffer
FUNCTION_BLOCK INTERNAL FB_BACnet_TLMBuffer EXTENDS FB_BACnet_BasePropertyLogBuffer
VAR PERSISTENT
	aBuffer : ARRAY[1 .. nBACnet_BufferSize] OF BYTE;
END_VAR
VAR CONSTANT
	{attribute 'hide'}
	{attribute 'parameterUnit':= 'byte'}
	nBACnet_HeaderSize		: UINT	:= 20;
	{attribute 'hide'}
	{attribute 'parameterUnit':= 'byte'}
	nBACnet_EntrySize		: UINT	:= 5;
	{attribute 'hide'}
	nBACnet_EntryCount		: UINT	:= BACnet_Globals.nDataField_MaxLogBufferEntries;
	{attribute 'hide'}
	nBACnet_EntryItemCount	: UINT	:= 100;
	
	{attribute 'hide'}
	nBACnet_BufferSize		: UINT	:= nBACnet_HeaderSize + ((nBACnet_EntrySize * nBACnet_EntryCount) * nBACnet_EntryItemCount);
END_VAR

SUPER^();

METHOD PROTECTED ValidateInst : BOOL
nBufferSize := SIZEOF(aBuffer);
pBufferValue := ADR(aBuffer);

ValidateInst := SUPER^.ValidateInst();
END_METHOD

METHOD FB_init : BOOL
VAR_INPUT
	bInitRetains : BOOL; // if TRUE, the retain variables are initialized (warm start / cold start)
	bInCopyCode : BOOL;  // if TRUE, the instance afterwards gets moved into the copy code (online change)
END_VAR
ePropertyID := E_BACnetPropIdentifier.PropLogBuffer;
END_METHOD

METHOD ResetValue
VAR
	stTimestamp : POINTER TO ST_BA_DateTime;
END_VAR
SUPER^.ResetValue();

// Write one log-entry "log-disabled" to buffer:
MemSetULINT(16#0000000100000020, nUsedSize);
MemSetUDINT(16#00000003, nUsedSize);

(*
stTimestamp := (pBufferValue+nUsedSize);
stTimestamp^ := F_GetCurrentTime();
nUsedSize := (nUsedSize+SIZEOF(ST_DateTime));
*)
MemSetULINT(16#51152607021D0177, nUsedSize);

MemSetUDINT(16#00000000, nUsedSize);
MemSetULINT(16#0000000000000008, nUsedSize);
MemSetULINT(16#0000800500000000, nUsedSize);
END_METHOD

END_FUNCTION_BLOCK

// POUs/Local/Objects/[Internal]/Property/Buffer/FB_BACnet_TrendLogBuffer
FUNCTION_BLOCK INTERNAL FB_BACnet_TrendLogBuffer EXTENDS FB_BACnet_BasePropertyLogBuffer
VAR PERSISTENT
	aBuffer : ARRAY[1 .. nBACnet_BufferSize] OF BYTE;
END_VAR
VAR CONSTANT
	{attribute 'parameterUnit':= 'byte'}
	nBACnet_EntrySize	: UINT	:= 56;
	nBACnet_EntryCount	: UINT	:= BACnet_Globals.nDataField_MaxLogBufferEntries;
	nBACnet_BufferSize	: UINT	:= (nBACnet_EntrySize * nBACnet_EntryCount);
END_VAR

SUPER^();

METHOD PROTECTED ValidateInst : BOOL
nBufferSize := SIZEOF(aBuffer);
pBufferValue := ADR(aBuffer);

ValidateInst := SUPER^.ValidateInst();
END_METHOD

METHOD FB_init : BOOL
VAR_INPUT
	bInitRetains : BOOL; // if TRUE, the retain variables are initialized (warm start / cold start)
	bInCopyCode : BOOL;  // if TRUE, the instance afterwards gets moved into the copy code (online change)
END_VAR
ePropertyID := E_BACnetPropIdentifier.PropLogBuffer;
END_METHOD

METHOD ResetValue
VAR
	stTimestamp : POINTER TO ST_BA_DateTime;
END_VAR
SUPER^.ResetValue();

// Write one log-entry "log-disabled" to buffer:
MemSetULINT(16#0000000100000020, nUsedSize);
MemSetUDINT(16#00000003, nUsedSize);

(*
stTimestamp := (pBufferValue+nUsedSize);
stTimestamp^ := F_GetCurrentTime();
nUsedSize := (nUsedSize+SIZEOF(ST_DateTime));
*)
MemSetULINT(16#51152607021D0177, nUsedSize);

MemSetUDINT(16#00000000, nUsedSize);
MemSetULINT(16#0000000000000008, nUsedSize);
MemSetULINT(16#0000800500000000, nUsedSize);
END_METHOD

END_FUNCTION_BLOCK

// POUs/Local/Objects/5P/FB_BACnet_AO_IO5P
// Analog Output Object
// - Terminal communication
// - 5 Priorities
{attribute 'pin_presentation_order_inputs' := 'bEnSfty,fValSfty,bEnCrit,fValCrit,bEnManLoc,fValManLoc,bEnPgm,fValPgm'}
{attribute 'pin_presentation_order_outputs' := 'fPresentValue,eActivePrio,bEvent,eReliability'}
FUNCTION_BLOCK FB_BACnet_AO_IO5P EXTENDS FB_BACnet_AO_IO
VAR_INPUT
	bEnSfty					: BOOL;
	fValSfty				: REAL;
	bEnCrit					: BOOL;
	fValCrit				: REAL;
	bEnManLoc				: BOOL;
	fValManLoc				: REAL;
END_VAR
VAR_INPUT CONSTANT PERSISTENT
	{region 'Operational Parameters'}
		{attribute 'parameterCategory':='Manual'}
		bEnManualRm : BOOL;
		{attribute 'parameterCategory':='Manual'}
		fValManualRm : REAL;
	{endregion}
END_VAR

SUPER^();

METHOD PROTECTED OnObjectStateChanged
SUPER^.OnObjectStateChanged();

CASE (tState) OF
	TCOM_STATE.TCOM_STATE_PREOP:
		// SyncHandler:
		RequestSyncHandlers(1, 4);
		
	TCOM_STATE.TCOM_STATE_SAFEOP:
		SyncPropertyPvPrio(E_BACnetPropIdentifier.PropPresentValue, SIZEOF(fValSfty), ADR(fValSfty), ADR(bEnSfty), BACnet_Param.ePrio_LifeSafety, 0, eFullSync_InitPLC, TRUE);
		SyncPropertyPvPrio(E_BACnetPropIdentifier.PropPresentValue, SIZEOF(fValCrit), ADR(fValCrit), ADR(bEnCrit), BACnet_Param.ePrio_Critical, 0, eFullSync_InitPLC, TRUE);
		SyncPropertyPvPrio(E_BACnetPropIdentifier.PropPresentValue, SIZEOF(fValManLoc), ADR(fValManLoc), ADR(bEnManLoc), BACnet_Param.ePrio_ManLocal, 0, eFullSync_InitPLC, TRUE);
		SyncPropertyPvPrio(E_BACnetPropIdentifier.PropPresentValue, SIZEOF(fValManualRm), ADR(fValManualRm), ADR(bEnManualRm), BACnet_Param.ePrio_ManRemote, 0, eFullSync_InitPLC, TRUE);
		
	TCOM_STATE.TCOM_STATE_OP:
		;
	
END_CASE
END_METHOD

PROPERTY EnManualRm : BOOL
GET
EnManualRm := bEnManualRm;
END_GET
SET
bEnManualRm := EnManualRm;
END_SET
END_PROPERTY

PROPERTY ValManualRm : REAL
GET
ValManualRm := fValManualRm;
END_GET
SET
fValManualRm := ValManualRm;
END_SET
END_PROPERTY

END_FUNCTION_BLOCK

// POUs/Local/Objects/FB_BACnet_AO_IO
// Analog Output Object
// - Terminal communication
// - 1 Priority
{attribute 'pin_presentation_order_outputs' := 'fPresentValue,bEvent,eReliability'}
FUNCTION_BLOCK FB_BACnet_AO_IO EXTENDS FB_BACnet_BaseAO
VAR_INPUT CONSTANT PERSISTENT
	{region 'Variable Parameters'}
		{attribute 'parameterCategory':='Config'}
		eOverriddenPolarity : E_BA_Polarity := E_BA_Polarity.eNormal;
	{endregion}
END_VAR
VAR
	{region 'Raw I/O'}
		bRawOverridden		AT %I*	: BOOL;				// Raw overridden (Optional)
		nRawState			AT %I*	: USINT;			// Raw state (Optional, only used to determine overridden state)
		nRawValue			AT %Q*	: INT;				// Raw value
	{endregion}
	{region 'Hardware'}
		_bIsOverriddenMapped		: BOOL;				// Indication to mapped hardware for overridden IO value
		_bIsStateMapped				: BOOL;				// Indication to mapped hardware for state
	{endregion}
END_VAR

IF (bReady) THEN
	// Overridden IO Value:
	IF (_bIsOverriddenMapped) THEN
		_bOverriddenValue := (bRawOverridden = (eOverriddenPolarity=E_BA_Polarity.eNormal));
	ELSIF (_bIsStateMapped) THEN
		_bOverriddenValue := ((nRawState=0) = (eOverriddenPolarity=E_BA_Polarity.eNormal));
	ELSE
		_bOverriddenValue := FALSE;
	END_IF
END_IF

SUPER^();

METHOD PROTECTED OnObjectStateChanged
SUPER^.OnObjectStateChanged();

CASE (tState) OF
	TCOM_STATE.TCOM_STATE_PREOP:
		// SyncHandler:
		RequestSyncHandlers(1, 0);

	TCOM_STATE.TCOM_STATE_SAFEOP:
		SyncProperty(E_BACnetPropIdentifier.PropRawIoAnalogValueINT, SIZEOF(nRawValue), ADR(nRawValue), 0, eSync_FromSupplement, TRUE);
		
	TCOM_STATE.TCOM_STATE_OP:
		// Check mapping of state:
		_bIsStateMapped := (F_GetMappingStatus(ADR(nRawState), SIZEOF(nRawState)) <> EPlcMappingStatus.MS_Unmapped);
		// Check mapping of overridden IO:
		_bIsOverriddenMapped := (F_GetMappingStatus(ADR(bRawOverridden), SIZEOF(bRawOverridden)) <> EPlcMappingStatus.MS_Unmapped);

END_CASE
END_METHOD

END_FUNCTION_BLOCK

// POUs/Local/Objects/5P/FB_BACnet_BO_IO5P
// Binary Output Object
// - Terminal communication
// - 5 Priorities
{attribute 'pin_presentation_order_inputs' := 'bEnSfty,bValSfty,bEnCrit,bValCrit,bEnManLoc,bValManLoc,bEnPgm,bValPgm'}
{attribute 'pin_presentation_order_outputs' := 'bPresentValue,eActivePrio,bEvent,eReliability'}
FUNCTION_BLOCK FB_BACnet_BO_IO5P EXTENDS FB_BACnet_BO_IO
VAR_INPUT
	bEnSfty					: BOOL;
	bValSfty				: BOOL;
	bEnCrit					: BOOL;
	bValCrit				: BOOL;
	bEnManLoc				: BOOL;
	bValManLoc				: BOOL;
END_VAR
VAR_INPUT CONSTANT PERSISTENT
	{region 'Operational Parameters'}
		{attribute 'parameterCategory':='Manual'}
		bEnManualRm : BOOL;
		{attribute 'parameterCategory':='Manual'}
		bValManualRm : BOOL;
	{endregion}
END_VAR

SUPER^();

METHOD PROTECTED OnObjectStateChanged
SUPER^.OnObjectStateChanged();

CASE (tState) OF
	TCOM_STATE.TCOM_STATE_PREOP:
		// SyncHandler:
		RequestSyncHandlers(1, 4);
		
	TCOM_STATE.TCOM_STATE_SAFEOP:
		SyncPropertyPvPrio(E_BACnetPropIdentifier.PropPresentValue, SIZEOF(bValSfty), ADR(bValSfty), ADR(bEnSfty), BACnet_Param.ePrio_LifeSafety, 0, eFullSync_InitPLC, TRUE);
		SyncPropertyPvPrio(E_BACnetPropIdentifier.PropPresentValue, SIZEOF(bValCrit), ADR(bValCrit), ADR(bEnCrit), BACnet_Param.ePrio_Critical, 0, eFullSync_InitPLC, TRUE);
		SyncPropertyPvPrio(E_BACnetPropIdentifier.PropPresentValue, SIZEOF(bValManLoc), ADR(bValManLoc), ADR(bEnManLoc), BACnet_Param.ePrio_ManLocal, 0, eFullSync_InitPLC, TRUE);
		SyncPropertyPvPrio(E_BACnetPropIdentifier.PropPresentValue, SIZEOF(bValManualRm), ADR(bValManualRm), ADR(bEnManualRm), BACnet_Param.ePrio_ManRemote, 0, eFullSync_InitPLC, TRUE);
		
	TCOM_STATE.TCOM_STATE_OP:
		;
		
END_CASE
END_METHOD

PROPERTY EnManualRm : BOOL
GET
EnManualRm := bEnManualRm;
END_GET
SET
bEnManualRm := EnManualRm;
END_SET
END_PROPERTY

PROPERTY ValManualRm : BOOL
GET
ValManualRm := bValManualRm;
END_GET
SET
bValManualRm := ValManualRm;
END_SET
END_PROPERTY

END_FUNCTION_BLOCK

// POUs/Local/Objects/FB_BACnet_BO_IO
// Binary Output Object
// - Terminal communication
// - 1 Priority
{attribute 'pin_presentation_order_outputs' := 'fPresentValue,bEvent,eReliability'}
FUNCTION_BLOCK FB_BACnet_BO_IO EXTENDS FB_BACnet_BaseBO
VAR_INPUT CONSTANT PERSISTENT
	{region 'Variable Parameters'}
		{attribute 'parameterCategory':='Config'}
		eFeedbackPolarity : E_BA_Polarity := E_BA_Polarity.eNormal;
		{attribute 'parameterCategory':='Config'}
		eOverriddenPolarity : E_BA_Polarity := E_BA_Polarity.eNormal;
	{endregion}
END_VAR
VAR
	{region 'Raw I/O'}
		bRawOverridden		AT %I*	: BOOL;				// Raw overridden (Optional)
		bRawValFeedback		AT %I*	: BOOL;				// Raw feedback Value (Optional)
		bRawValue			AT %Q*	: BOOL;				// Raw value
	{endregion}
	{region 'Hardware'}
		_bIsFeedbackMapped			: BOOL;				// Indication to mapped hardware for feedback value
		_bIsOverriddenMapped		: BOOL;				// Indication to mapped hardware for overridden IO value
	{endregion}
	{region 'Internal'}
		_bOverriddenValue			: BOOL;
	{endregion}
END_VAR
VAR_STAT 
	// (BETA) ... Following symbols should be made non-static / thread safe!
	{region 'Temporary'}
		{attribute 'hide'}
		_bEnFeedback				: BOOL;
	{endregion}
END_VAR

IF (bReady) THEN
	// Overridden IO Value:
	_bOverriddenValue := SEL(_bIsOverriddenMapped, FALSE, (bRawOverridden = (eOverriddenPolarity=E_BA_Polarity.eNormal)));
	
	// Feedback Value:
	_bEnFeedback := SEL(_bIsFeedbackMapped, FALSE, NOT _bOverriddenValue);
	_bFeedbackValue := SEL(_bEnFeedback, bPresentValue, (bRawValFeedback = (eFeedbackPolarity=E_BA_Polarity.eNormal)));
END_IF

SUPER^();

METHOD PROTECTED OnObjectStateChanged
SUPER^.OnObjectStateChanged();

CASE (tState) OF
	TCOM_STATE.TCOM_STATE_PREOP:
		// SyncHandler:
		RequestSyncHandlers(1, 1);

	TCOM_STATE.TCOM_STATE_SAFEOP:
		SyncProperty(E_BACnetPropIdentifier.PropRawIoBinaryValueBOOL, SIZEOF(bRawValue), ADR(bRawValue), 0, eSync_FromSupplement, TRUE);
		
	TCOM_STATE.TCOM_STATE_OP:
		SyncProperty(E_BACnetPropIdentifier.PropRawIoStateOverrideInverted, SIZEOF(_bOverriddenValue), ADR(_bOverriddenValue), 0, eSync_ToSupplement, FALSE);

		// Check mapping of feedback:
		_bIsFeedbackMapped := (F_GetMappingStatus(ADR(bRawValFeedback), SIZEOF(bRawValFeedback)) <> EPlcMappingStatus.MS_Unmapped);
		// Check mapping of overridden IO:
		_bIsOverriddenMapped := (F_GetMappingStatus(ADR(bRawOverridden), SIZEOF(bRawOverridden)) <> EPlcMappingStatus.MS_Unmapped);
		
END_CASE
END_METHOD

END_FUNCTION_BLOCK

// POUs/Local/Objects/5P/FB_BACnet_MO_IO5P
// Multistate Output Object
// - Terminal communication
// - 5 Priorities
{attribute 'pin_presentation_order_inputs' := 'bEnSfty,nValSfty,bEnCrit,nValCrit,bEnManLoc,nValManLoc,bEnPgm,nValPgm'}
{attribute 'pin_presentation_order_outputs' := 'nPresentValue,eActivePrio,bEvent,eReliability'}
FUNCTION_BLOCK FB_BACnet_MO_IO5P EXTENDS FB_BACnet_MO_IO
VAR_INPUT
	bEnSfty					: BOOL;
	nValSfty				: UDINT		:= 1;
	bEnCrit					: BOOL;
	nValCrit				: UDINT		:= 1;
	bEnManLoc				: BOOL;
	nValManLoc				: UDINT		:= 1;
END_VAR
VAR_INPUT CONSTANT PERSISTENT
	{region 'Operational Parameters'}
		{attribute 'parameterCategory':='Manual'}
		bEnManualRm : BOOL;
		{attribute 'parameterCategory':='Manual'}
		nValManualRm : UDINT := 1;
	{endregion}
END_VAR

SUPER^();

METHOD PROTECTED OnObjectStateChanged
SUPER^.OnObjectStateChanged();

CASE (tState) OF
	TCOM_STATE.TCOM_STATE_PREOP:
		// SyncHandler:
		RequestSyncHandlers(1, 4);
		
	TCOM_STATE.TCOM_STATE_SAFEOP:
		SyncPropertyPvPrio(E_BACnetPropIdentifier.PropPresentValue, SIZEOF(nValSfty), ADR(nValSfty), ADR(bEnSfty), BACnet_Param.ePrio_LifeSafety, 0, eFullSync_InitPLC, TRUE);
		SyncPropertyPvPrio(E_BACnetPropIdentifier.PropPresentValue, SIZEOF(nValCrit), ADR(nValCrit), ADR(bEnCrit), BACnet_Param.ePrio_Critical, 0, eFullSync_InitPLC, TRUE);
		SyncPropertyPvPrio(E_BACnetPropIdentifier.PropPresentValue, SIZEOF(nValManLoc), ADR(nValManLoc), ADR(bEnManLoc), BACnet_Param.ePrio_ManLocal, 0, eFullSync_InitPLC, TRUE);
		SyncPropertyPvPrio(E_BACnetPropIdentifier.PropPresentValue, SIZEOF(nValManualRm), ADR(nValManualRm), ADR(bEnManualRm), BACnet_Param.ePrio_ManRemote, 0, eFullSync_InitPLC, TRUE);
		
	TCOM_STATE.TCOM_STATE_OP:
		;
		
END_CASE
END_METHOD

PROPERTY EnManualRm : BOOL
GET
EnManualRm := bEnManualRm;
END_GET
SET
bEnManualRm := EnManualRm;
END_SET
END_PROPERTY

PROPERTY ValManualRm : UDINT
GET
ValManualRm := nValManualRm;
END_GET
SET
nValManualRm := ValManualRm;
END_SET
END_PROPERTY

END_FUNCTION_BLOCK

// POUs/Local/Objects/FB_BACnet_MO_IO
// Multistate Output Object
// - Terminal communication
// - 1 Priority
{attribute 'pin_presentation_order_outputs' := 'fPresentValue,bEvent,eReliability'}
FUNCTION_BLOCK FB_BACnet_MO_IO EXTENDS FB_BACnet_BaseMO
VAR_INPUT CONSTANT PERSISTENT
	{region 'Variable Parameters'}
		{attribute 'parameterCategory':='Config'}
		eMappingMode : E_BA_ByteMappingMode := E_BA_ByteMappingMode.eIndex1N;
		{attribute 'parameterCategory':='Config'}
		eFeedbackMappingMode : E_BA_ByteMappingMode := E_BA_ByteMappingMode.eIndex1N;
	{endregion}
END_VAR
VAR
	{region 'Raw I/O'}
		bRawValFeedback		AT %I*	: ST_BA_Byte;		// Bus terminal feedback Value (Optional)
		bRawValue			AT %Q*	: ST_BA_Byte;		// Bus terminal value
	{endregion}
	{region 'Hardware'}
		_bIsFeedbackMapped			: BOOL;				// Indication to mapped hardware for feedback value
	{endregion}
	{region 'Internal'}
		nLastPresentValue			: UDINT;
	{endregion}
END_VAR

IF (bReady) THEN
	// Feedback Value:
	IF (_bIsFeedbackMapped) THEN
		F_BA_MapUDIFromRawByte(_nFeedbackValue, ADR(bRawValFeedback), eFeedbackMappingMode, nRelinquishDefault);
	ELSE
		_nFeedbackValue := nPresentValue;
	END_IF
	
	// Trigger change of value:
	IF (nPresentValue <> nLastPresentValue) THEN
		nLastPresentValue := nPresentValue;
		F_BA_MapUDIToRawByte(nPresentValue, ADR(bRawValue), eMappingMode, nRelinquishDefault);
	END_IF
ELSE
	nPresentValue := nRelinquishDefault;
	
	// Set last value to a different value compared to actual raw value (So a COV is triggered when current instance becomes ready):
	nLastPresentValue := (nLastPresentValue+1);
END_IF

SUPER^();

METHOD PROTECTED OnObjectStateChanged
SUPER^.OnObjectStateChanged();

CASE (tState) OF
	TCOM_STATE.TCOM_STATE_PREOP:
		;

	TCOM_STATE.TCOM_STATE_SAFEOP:
		;
		
	TCOM_STATE.TCOM_STATE_OP:
		// Check mapping of feedback:
		_bIsFeedbackMapped := (F_GetMappingStatus(ADR(bRawValFeedback), SIZEOF(bRawValFeedback)) <> EPlcMappingStatus.MS_Unmapped);
		
END_CASE
END_METHOD

END_FUNCTION_BLOCK

// POUs/Local/Objects/Experimental/FB_BACnet_ExpTLM
{attribute 'hide'}	// (BETA) ...FB is only for testing!


FUNCTION_BLOCK FB_BACnet_ExpTLM EXTENDS FB_BACnet_BaseTLog
VAR_INPUT CONSTANT PERSISTENT
	{region 'Fixed Parameters'}
		// (BETA) ... Implement "LogBuffer(Multiple)"-Property
		//{attribute 'hide'}
		//{attribute 'parameterCategory':='Value'}
		//aLogBuffer : ARRAY [1 .. BACnet_Param.nTLM_ArraySize] OF ST_BACnet_TLMEntry;
	{endregion}
END_VAR
VAR PERSISTENT
	{region 'SubInit'}
		// (BETA) ... Implement "DeviceObjPropRef(Multiple)"-Property
		// ...
	{endregion}
END_VAR
VAR
	{region 'Buffers'}
		{attribute 'conditionalshow'}
		fbLogBuffer					: FB_BACnet_TLMBuffer			:= (iRefObject := THIS^);
	{endregion}
END_VAR

// Synchronize Buffers:
fbLogBuffer();

SUPER^();

METHOD PROTECTED OnObjectStateChanged
SUPER^.OnObjectStateChanged();

// Synchronize:
fbLogBuffer.OnObjectStateChanged(tState);

CASE (tState) OF
	TCOM_STATE.TCOM_STATE_PREOP:
		;
	
	TCOM_STATE.TCOM_STATE_SAFEOP:
		;

	TCOM_STATE.TCOM_STATE_OP:
		;
		
END_CASE
END_METHOD

METHOD FB_init : BOOL
VAR_INPUT
	bInitRetains : BOOL; // if TRUE, the retain variables are initialized (warm start / cold start)
	bInCopyCode : BOOL;  // if TRUE, the instance afterwards gets moved into the copy code (online change)
END_VAR
eObjectType := E_BACnetObjType.ObjTrendLogMultiple;
END_METHOD

END_FUNCTION_BLOCK

// POUs/Local/Objects/Experimental/FB_BACnet_ExpTLog
{attribute 'hide'}	// (BETA) ...FB is only for testing!



FUNCTION_BLOCK FB_BACnet_ExpTLog EXTENDS FB_BACnet_BaseTLog

// (BETA) ... Implement "LogBuffer"-Property
///////////////////////////////////////////////////////////////
VAR_INPUT CONSTANT
	bTrendLog_Write	: BOOL;
END_VAR
///////////////////////////////////////////////////////////////


VAR_INPUT CONSTANT PERSISTENT
	{region 'Variable Parameters'}
		{attribute 'parameterCategory':='Value'}
		aLogBuffer : T_BACnet_TLogBuffer;
			 
		{attribute 'parameterCategory':='Config'}
		stObjectPropertyReference : ST_BACnet_ObjectPropertyReference;
	{endregion}
END_VAR
VAR
	{region 'Buffers'}
		{attribute 'conditionalshow'}
		fbLogBuffer					: FB_BACnet_TrendLogBuffer			:= (iRefObject := THIS^);
	{endregion}
	{region 'Internal'}
		bLogBufferChanged			: BOOL;
	{endregion}
END_VAR

// Synchronize Buffers:
fbLogBuffer();

// (BETA) ... Implement "LogBuffer"-Property
///////////////////////////////////////////////////////////////
IF bTrendLog_Write THEN
	bTrendLog_Write := FALSE;
	{warning disable C0196}
	WritePropertyLogBuffer(aLogBuffer);
	{warning restore C0196}
END_IF
///////////////////////////////////////////////////////////////

IF bLogBufferChanged THEN
	bLogBufferChanged := FALSE;
	{warning disable C0196}
	ReadPropertyLogBuffer(aLogBuffer);
	{warning restore C0196}
END_IF

SUPER^();

METHOD PROTECTED OnObjectStateChanged
SUPER^.OnObjectStateChanged();

// Synchronize:
fbLogBuffer.OnObjectStateChanged(tState);

CASE (tState) OF
	TCOM_STATE.TCOM_STATE_PREOP:
		;
	
	TCOM_STATE.TCOM_STATE_SAFEOP:
		;

	TCOM_STATE.TCOM_STATE_OP:
		// Validate referred property:
		IF (ValidateReference(stObjectPropertyReference.iObject, stObjectPropertyReference.tObjectID, 16#FF)) THEN
			ObjectPropertyReference := stObjectPropertyReference;
		END_IF
		
END_CASE
END_METHOD

METHOD FB_init : BOOL
VAR_INPUT
	bInitRetains : BOOL; // if TRUE, the retain variables are initialized (warm start / cold start)
	bInCopyCode : BOOL;  // if TRUE, the instance afterwards gets moved into the copy code (online change)
END_VAR
eObjectType := E_BACnetObjType.ObjTrendLog;
END_METHOD

PROPERTY ObjectPropertyReference : ST_BACnet_ObjectPropertyReference
GET
ObjectPropertyReference := stObjectPropertyReference;
END_GET
SET
stObjectPropertyReference := ObjectPropertyReference;

WritePropertyReference(E_BACnetPropIdentifier.PropLogDeviceObjectProperty, stObjectPropertyReference);
END_SET
END_PROPERTY

END_FUNCTION_BLOCK

// POUs/Local/Objects/FB_BACnet_AI
// Analog Input Object
// - process value
{attribute 'pin_presentation_order_outputs' := 'fPresentValue,bEvent,eReliability'}
{attribute 'enable_dynamic_creation'}
FUNCTION_BLOCK FB_BACnet_AI EXTENDS FB_BACnet_BaseAI
VAR_INPUT
	fVal						: REAL;				// Process value
END_VAR

IF bReady THEN
	IF NOT bOutOfService THEN
		fPresentValue := fVal;
	END_IF
ELSE
	fPresentValue := 0;
END_IF

SUPER^();

METHOD PROTECTED OnObjectStateChanged
CASE (tState) OF
	TCOM_STATE.TCOM_STATE_PREOP:
		// SyncHandler:
		RequestSyncHandlers(0, 1);
		
		// Properties:
		EnableProperty(E_BACnetPropIdentifier.PropResolution, FALSE);
		EnableProperty(E_BACnetPropIdentifier.PropScaleOffset, FALSE);

	TCOM_STATE.TCOM_STATE_SAFEOP:
		SyncProperty(E_BACnetPropIdentifier.PropPresentValue, SIZEOF(fPresentValue), ADR(fPresentValue), 0, eFullSync_InitPLC, TRUE);
		
	TCOM_STATE.TCOM_STATE_OP:
		;

END_CASE

SUPER^.OnObjectStateChanged();
END_METHOD

END_FUNCTION_BLOCK

// POUs/Local/Objects/FB_BACnet_AI_IO
// Analog Input Object
// - Terminal communication
{attribute 'pin_presentation_order_outputs' := 'fPresentValue,bEvent,eReliability'}
FUNCTION_BLOCK FB_BACnet_AI_IO EXTENDS FB_BACnet_BaseAI
VAR_INPUT CONSTANT PERSISTENT	
	{region 'Variable Parameters'}
		{attribute 'parameterCategory':='Hardware'}
		fResolution : REAL := 0.1;
		{attribute 'parameterCategory':='Hardware'}
		fScaleOffset : REAL := 0;
	{endregion}
END_VAR
VAR
	{region 'Raw I/O'}
		nRawState			AT %I*	: USINT;			// Bus terminal state
		nRawValue			AT %I*	: INT;				// Bus terminal value
	{endregion}
END_VAR

SUPER^();

METHOD PROTECTED OnObjectStateChanged
CASE (tState) OF
	TCOM_STATE.TCOM_STATE_PREOP:
		// SyncHandler:
		RequestSyncHandlers(1, 4);

	TCOM_STATE.TCOM_STATE_SAFEOP:
		SyncProperty(E_BACnetPropIdentifier.PropPresentValue, SIZEOF(fPresentValue), ADR(fPresentValue), 0, eSync_FromSupplement, TRUE);
		
		SyncProperty(E_BACnetPropIdentifier.PropRawIoStateUSINT, SIZEOF(nRawState), ADR(nRawState), 0, eSync_ToSupplement, TRUE);
		SyncProperty(E_BACnetPropIdentifier.PropRawIoAnalogValueINT, SIZEOF(nRawValue), ADR(nRawValue), 0, eSync_ToSupplement, TRUE);
		
	TCOM_STATE.TCOM_STATE_OP:
		SyncProperty(E_BACnetPropIdentifier.PropResolution, SIZEOF(fResolution), ADR(fResolution), 0, eFullSync_InitPLC, FALSE);
		SyncProperty(E_BACnetPropIdentifier.PropScaleOffset, SIZEOF(fScaleOffset), ADR(fScaleOffset), 0, eFullSync_InitPLC, FALSE);

END_CASE

SUPER^.OnObjectStateChanged();
END_METHOD

END_FUNCTION_BLOCK

// POUs/Local/Objects/FB_BACnet_BI_IO
// Binary Input Object
// - Terminal communication
{attribute 'pin_presentation_order_outputs' := 'bPresentValue,bEvent,eReliability'}
FUNCTION_BLOCK FB_BACnet_BI_IO EXTENDS FB_BACnet_BaseBI
VAR
	{region 'Raw I/O'}
		bRawValue			AT %I*	: BOOL;				// Bus terminal value
	{endregion}
END_VAR

SUPER^();

METHOD PROTECTED OnObjectStateChanged
SUPER^.OnObjectStateChanged();

CASE (tState) OF
	TCOM_STATE.TCOM_STATE_PREOP:
		// SyncHandler:
		RequestSyncHandlers(0, 1);

	TCOM_STATE.TCOM_STATE_SAFEOP:
		SyncProperty(E_BACnetPropIdentifier.PropRawIoBinaryValueBOOL, SIZEOF(bRawValue), ADR(bRawValue), 0, eSync_ToSupplement, TRUE);
		
	TCOM_STATE.TCOM_STATE_OP:
		;

END_CASE
END_METHOD

END_FUNCTION_BLOCK

// POUs/Local/Objects/FB_BACnet_EE
// Calendar Object
{attribute 'enable_dynamic_creation'}
FUNCTION_BLOCK FB_BACnet_EE EXTENDS FB_BACnet_EventObject 
VAR_INPUT CONSTANT PERSISTENT
	{region 'Variable Parameters'}
		{attribute 'parameterCategory':='Value'}
		stEventParameter : ST_BACnet_EventParameter;
		{attribute 'parameterCategory':='Config'}
		stObjectPropertyReference : ST_BACnet_ObjectPropertyReference;
	{endregion}
END_VAR
VAR_INPUT CONSTANT
	{region 'Variable Parameters'}
		{attribute 'parameterCategory':='Value'}
		bWriteEventParameter : BOOL;
	{endregion}
END_VAR
VAR	
	{region 'COV'}
		bEventParameterChanged	: BOOL;
	{endregion}
END_VAR

IF (bWriteEventParameter) THEN
	WriteContent();
	bWriteEventParameter := FALSE;
END_IF
IF (bEventParameterChanged) THEN
	ReadContent();
	bEventParameterChanged := FALSE;
END_IF

SUPER^();

METHOD PROTECTED OnObjectStateChanged
SUPER^.OnObjectStateChanged();

CASE (tState) OF
	TCOM_STATE.TCOM_STATE_PREOP:
		// SyncHandler:
		RequestSyncHandlers(1, 0);

	TCOM_STATE.TCOM_STATE_SAFEOP:
		;
		
	TCOM_STATE.TCOM_STATE_OP:
		// Validate referred property:
		IF (ValidateReference(stObjectPropertyReference.iObject, stObjectPropertyReference.tObjectID, 16#FF)) THEN
			ObjectPropertyReference := stObjectPropertyReference;
		END_IF
	
		SyncPropertyCOV(E_BACnetPropIdentifier.PropEventParameters, ADR(bEventParameterChanged));
		WriteContent();	
END_CASE
END_METHOD

METHOD FB_init : BOOL
VAR_INPUT
	bInitRetains : BOOL; // if TRUE, the retain variables are initialized (warm start / cold start)
	bInCopyCode : BOOL;  // if TRUE, the instance afterwards gets moved into the copy code (online change)
END_VAR
eObjectType := E_BACnetObjType.ObjEventEnrollment;
END_METHOD

METHOD ReadContent : BOOL
ReadContent := (ReadPropertyEventParameter(stEventParameter) = S_OK);
END_METHOD

METHOD WriteContent : BOOL
WriteContent := (WritePropertyEventParameter(stEventParameter) = S_OK);
END_METHOD

PROPERTY ObjectPropertyReference : ST_BACnet_ObjectPropertyReference
GET
ObjectPropertyReference := stObjectPropertyReference;
END_GET
SET
stObjectPropertyReference := ObjectPropertyReference;

WritePropertyReference(E_BACnetPropIdentifier.PropObjectPropertyReference, stObjectPropertyReference);
END_SET
END_PROPERTY

END_FUNCTION_BLOCK

// POUs/Local/Objects/FB_BACnet_EventLog
// Event Log Object
FUNCTION_BLOCK FB_BACnet_EventLog EXTENDS FB_BACnet_Object
VAR_INPUT CONSTANT PERSISTENT
	{region 'Fixed Parameters'}
		{attribute 'parameterCategory':='Value'}
		nBufferSize : UDINT := BACnet_Param.nEventLog_ArraySize;
		// (BETA) ... Implement "EventLogBuffer"-Property
		//{attribute 'hide'}
		//{attribute 'parameterCategory':='Value'}
		//aLogBuffer : ARRAY [1 .. BACnet_Param.nEventLog_ArraySize] OF ST_BACnet_EventLogEntry;
			 
		{attribute 'parameterCategory':='Config'}
		nProcessId : UDINT;
	{endregion}
	{region 'Variable Parameters'}
		{attribute 'parameterCategory':='State'}
		bLogEnable : BOOL;
			 
		{attribute 'parameterCategory':='EventConfig'}
		nNotificationClass : UDINT;
		{attribute 'parameterCategory':='EventConfig'}
		eNotifyType : E_BACnet_NotifyType := E_BACnet_NotifyType.eAlarm;
		{attribute 'parameterCategory':='EventConfig'}
		aEventEnable : T_BACnet_EventTransitions;
		{attribute 'parameterCategory':='EventConfig'}
		aEventMessageTextsConfig : T_BACnet_EventTransitionTexts;
		
		{attribute 'parameterCategory':='Config'}
		stStartTime : ST_BA_DateTime;
		{attribute 'parameterCategory':='Config'}
		stStopTime : ST_BA_DateTime;
		{attribute 'parameterCategory':='Config'}
		bStopWhenFull : BOOL;
		{attribute 'parameterCategory':='Config'}
		nNotificationThreshold : UDINT := 50;
	{endregion}
END_VAR
VAR_OUTPUT
	nRecordCount				: UDINT;
	nTotalRecordCount			: UDINT;
END_VAR
VAR
	{region 'Buffers'}
		{attribute 'conditionalshow'}
		fbLogBuffer				: FB_BACnet_EventLogBuffer	:= (iRefObject := THIS^);
	{endregion}
END_VAR

// Synchronize Buffers:
fbLogBuffer();

SUPER^();

METHOD PROTECTED OnObjectStateChanged
SUPER^.OnObjectStateChanged();

CASE (tState) OF
	TCOM_STATE.TCOM_STATE_PREOP:
		// SyncHandler:
		RequestSyncHandlers(2, 14);
		
		// Properties:
		// May limit buffer size to respect array size:
		nBufferSize := MIN(BACnet_Param.nEventLog_ArraySize, nBufferSize);
		
		WritePropertyUDInt(E_BACnetPropIdentifier.PropBufferSize, nBufferSize);
		
		// Ensure UTF-8 Encoding:
		F_BA_EnsureUTF8Array(ADR(aEventMessageTextsConfig), SIZEOF(aEventMessageTextsConfig[1]), TO_DINT(E_BA_EventTransition.Count));
		
		IF nProcessId = 0 THEN
			EnableProperty(E_BACnetPropIdentifier.PropProcessId, FALSE);
		END_IF
		
	TCOM_STATE.TCOM_STATE_SAFEOP:
		;

	TCOM_STATE.TCOM_STATE_OP:
		ConcatTitle(aEventMessageTextsConfig[E_BA_EventTransition.eToOffnormal], sDescription, BACnet_Param.sSeparator_EventMessageText);
		ConcatTitle(aEventMessageTextsConfig[E_BA_EventTransition.eToFault], sDescription, BACnet_Param.sSeparator_EventMessageText);
		ConcatTitle(aEventMessageTextsConfig[E_BA_EventTransition.eToNormal], sDescription, BACnet_Param.sSeparator_EventMessageText);
		
		// Synchronize:
		SyncProperty(E_BACnetPropIdentifier.PropRecordCount, SIZEOF(nRecordCount), ADR(nRecordCount), 0, eSync_FromSupplement, FALSE);
		SyncProperty(E_BACnetPropIdentifier.PropTotalRecordCount, SIZEOF(nTotalRecordCount), ADR(nTotalRecordCount), 0, eSync_FromSupplement, FALSE);
		
		SyncProperty(E_BACnetPropIdentifier.PropNotificationClass, SIZEOF(nNotificationClass), ADR(nNotificationClass), 0, eFullSync_InitPLC, FALSE);
		SyncProperty(E_BACnetPropIdentifier.PropNotifyType, SIZEOF(eNotifyType), ADR(eNotifyType), 0, eFullSync_InitPLC, FALSE);
		SyncPropertyIdx(E_BACnetPropIdentifier.PropEventEnable, SIZEOF(BOOL), ADR(aEventEnable[E_BA_EventTransition.eToOffnormal]), E_BACnet_EventTransitionBits.eToOffnormal, 0, eFullSync_InitPLC, FALSE);	
		SyncPropertyIdx(E_BACnetPropIdentifier.PropEventEnable, SIZEOF(BOOL), ADR(aEventEnable[E_BA_EventTransition.eToFault]), E_BACnet_EventTransitionBits.eToFault, 0, eFullSync_InitPLC, FALSE);	
		SyncPropertyIdx(E_BACnetPropIdentifier.PropEventEnable, SIZEOF(BOOL), ADR(aEventEnable[E_BA_EventTransition.eToNormal]), E_BACnet_EventTransitionBits.eToNormal, 0, eFullSync_InitPLC, FALSE);
		SyncPropertyIdx(E_BACnetPropIdentifier.PropEventMessageTextsConfig, SIZEOF(T_MaxString), ADR(aEventMessageTextsConfig[E_BA_EventTransition.eToOffnormal]), (E_BACnet_EventTransitionBits.eToOffnormal+1), 0, eFullSync_InitPLC, FALSE);
		SyncPropertyIdx(E_BACnetPropIdentifier.PropEventMessageTextsConfig, SIZEOF(T_MaxString), ADR(aEventMessageTextsConfig[E_BA_EventTransition.eToFault]), (E_BACnet_EventTransitionBits.eToFault+1), 0, eFullSync_InitPLC, FALSE);
		SyncPropertyIdx(E_BACnetPropIdentifier.PropEventMessageTextsConfig, SIZEOF(T_MaxString), ADR(aEventMessageTextsConfig[E_BA_EventTransition.eToNormal]), (E_BACnet_EventTransitionBits.eToNormal+1), 0, eFullSync_InitPLC, FALSE);
		
		SyncProperty(E_BACnetPropIdentifier.PropEnable, SIZEOF(bLogEnable), ADR(bLogEnable), 0, eFullSync_InitPLC, FALSE);
		SyncProperty(E_BACnetPropIdentifier.PropStartTime, SIZEOF(stStartTime), ADR(stStartTime), 0, eFullSync_InitPLC, FALSE);
		SyncProperty(E_BACnetPropIdentifier.PropStopTime, SIZEOF(stStopTime), ADR(stStopTime), 0, eFullSync_InitPLC, FALSE);
		SyncProperty(E_BACnetPropIdentifier.PropStopWhenFull, SIZEOF(bStopWhenFull), ADR(bStopWhenFull), 0, eFullSync_InitPLC, FALSE);
		SyncProperty(E_BACnetPropIdentifier.PropNotificationThreshold, SIZEOF(nNotificationThreshold), ADR(nNotificationThreshold), 0, eFullSync_InitPLC, FALSE);
		IF nProcessId <> 0 THEN
			SyncProperty(E_BACnetPropIdentifier.PropProcessId, SIZEOF(nProcessId), ADR(nProcessId), 0, eFullSync_InitPLC, FALSE);
		END_IF
END_CASE

// Synchronize:
fbLogBuffer.OnObjectStateChanged(tState);
END_METHOD

METHOD FB_init : BOOL
VAR_INPUT
	bInitRetains : BOOL; // if TRUE, the retain variables are initialized (warm start / cold start)
	bInCopyCode : BOOL;  // if TRUE, the instance afterwards gets moved into the copy code (online change)
END_VAR
eObjectType := E_BACnetObjType.ObjEventLog;
END_METHOD

END_FUNCTION_BLOCK

// POUs/Local/Objects/FB_BACnet_MI_IO
// Multistate Input Object
// - Terminal communication
{attribute 'pin_presentation_order_outputs' := 'nPresentValue,bEvent,eReliability'}
FUNCTION_BLOCK FB_BACnet_MI_IO EXTENDS FB_BACnet_BaseMI
VAR_INPUT CONSTANT PERSISTENT
	{region 'Variable Parameters'}
		{attribute 'parameterCategory':='Config'}
		eMappingMode : E_BA_ByteMappingMode := E_BA_ByteMappingMode.eIndex1N;
		
		// Used value when no raw-value is active.
		// Note: The mapped process value is shifted '+1' when it is higher than this default value.
		//       > In fact the default value sorts into the range of valid process values.
		{attribute 'parameterCategory':='Value'}
		nRelinquishDefault : UDINT := 1;
	{endregion}
END_VAR
VAR
	{region 'Raw I/O'}
		bRawValue		AT %I*	: ST_BA_Byte;				// Bus terminal value
	{endregion}
	{region 'Internal'}
		bLastRawValue			: BYTE;
	{endregion}
END_VAR
VAR_STAT
	// (BETA) ... Following symbols should be made non-static / thread safe!
	{region 'Temporary'}
		{attribute 'hide'}
		_bRawValue				: POINTER TO BYTE;
	{endregion}
END_VAR

_bRawValue := ADR(bRawValue);

IF bReady THEN	
	// Trigger change of value:
	IF (_bRawValue^ <> bLastRawValue) THEN
		bLastRawValue := _bRawValue^;
		F_BA_MapUDIFromRawByte(nPresentValue, ADR(bRawValue), eMappingMode, nRelinquishDefault);
	END_IF
ELSE
	// Set last value to a different value compared to actual raw value (So a COV is triggered when current instance becomes ready):
	bLastRawValue := (_bRawValue^+1);
	
	nPresentValue := nRelinquishDefault;
END_IF

SUPER^();

END_FUNCTION_BLOCK

// POUs/Local/Objects/FB_BACnet_TLM
FUNCTION_BLOCK FB_BACnet_TLM EXTENDS FB_BACnet_BaseTLog
VAR_INPUT CONSTANT PERSISTENT
	{region 'Variable Parameters'}
		{attribute 'parameterCategory':='Config'}
		aObjectPropertyReferences : T_BACnet_ObjectPropertyReferenceList;
	{endregion}
END_VAR
VAR
	{region 'Buffers'}
		{attribute 'conditionalshow'}
		fbLogBuffer					: FB_BACnet_TLMBuffer			:= (iRefObject := THIS^);
	{endregion}
END_VAR

// Synchronize Buffers:
fbLogBuffer();

SUPER^();

METHOD PROTECTED OnObjectStateChanged
VAR
	i : DINT;
	_bResult : BOOL;
END_VAR
SUPER^.OnObjectStateChanged();

CASE (tState) OF
	TCOM_STATE.TCOM_STATE_PREOP:
		;
	TCOM_STATE.TCOM_STATE_SAFEOP:
		;
	TCOM_STATE.TCOM_STATE_OP:
		// Validate referred properties:
		FOR i:= 1 TO TO_DINT(BACnet_Param.nRefList_ReferenceCount) DO
			ValidateReference(aObjectPropertyReferences[i].iObject, aObjectPropertyReferences[i].tObjectID, 16#FF);
		END_FOR
		ObjectPropertyReferences := aObjectPropertyReferences;
END_CASE


// Synchronize:
fbLogBuffer.OnObjectStateChanged(tState);
END_METHOD

METHOD FB_init : BOOL
VAR_INPUT
	bInitRetains : BOOL; // if TRUE, the retain variables are initialized (warm start / cold start)
	bInCopyCode : BOOL;  // if TRUE, the instance afterwards gets moved into the copy code (online change)
END_VAR
eObjectType := E_BACnetObjType.ObjTrendLogMultiple;
END_METHOD

PROPERTY ObjectPropertyReferences : T_BACnet_ObjectPropertyReferenceList
GET
ObjectPropertyReferences := aObjectPropertyReferences;
END_GET
SET
aObjectPropertyReferences := ObjectPropertyReferences;

WritePropertyReferenceList(E_BACnetPropIdentifier.PropLogDeviceObjectProperty, aObjectPropertyReferences);
END_SET
END_PROPERTY

END_FUNCTION_BLOCK

// POUs/Local/Objects/FB_BACnet_TLog
FUNCTION_BLOCK FB_BACnet_TLog EXTENDS FB_BACnet_BaseTLog
VAR_INPUT CONSTANT PERSISTENT
	{region 'Variable Parameters'}
		{attribute 'parameterCategory':='Config'}
		stObjectPropertyReference : ST_BACnet_ObjectPropertyReference;
	{endregion}
END_VAR
VAR
	{region 'Buffers'}
		{attribute 'conditionalshow'}
		fbLogBuffer					: FB_BACnet_TrendLogBuffer			:= (iRefObject := THIS^);
	{endregion}
END_VAR

// Synchronize Buffers:
fbLogBuffer();

SUPER^();

METHOD PROTECTED OnObjectStateChanged
SUPER^.OnObjectStateChanged();

CASE (tState) OF
	TCOM_STATE.TCOM_STATE_PREOP:
		;
	TCOM_STATE.TCOM_STATE_SAFEOP:
		;
	TCOM_STATE.TCOM_STATE_OP:
		// Validate referred property:
		IF (ValidateReference(stObjectPropertyReference.iObject, stObjectPropertyReference.tObjectID, 16#FF)) THEN
			ObjectPropertyReference := stObjectPropertyReference;
		END_IF
		
END_CASE


fbLogBuffer.OnObjectStateChanged(tState);
END_METHOD

METHOD FB_init : BOOL
VAR_INPUT
	bInitRetains : BOOL; // if TRUE, the retain variables are initialized (warm start / cold start)
	bInCopyCode : BOOL;  // if TRUE, the instance afterwards gets moved into the copy code (online change)
END_VAR
eObjectType := E_BACnetObjType.ObjTrendLog;
END_METHOD

PROPERTY ObjectPropertyReference : ST_BACnet_ObjectPropertyReference
GET
ObjectPropertyReference := stObjectPropertyReference;
END_GET
SET
stObjectPropertyReference := ObjectPropertyReference;

WritePropertyReference(E_BACnetPropIdentifier.PropLogDeviceObjectProperty, stObjectPropertyReference);
END_SET
END_PROPERTY

END_FUNCTION_BLOCK

// POUs/Remote/Objects/Basic/[Base]/Basic/FB_BACnetRM_Object
FUNCTION_BLOCK FB_BACnetRM_Object EXTENDS FB_BACnetRM_BaseObject IMPLEMENTS I_BACnetRM_Object, I_BACnetRM_ObjectOwner
VAR
	{region 'Internal'}
		{attribute 'hide'}
		bParentInit					: BOOL := TRUE;
		{attribute 'hide'}
		fbLogMsg					: FB_BA_LogMessage;
	{endregion}
END_VAR

SUPER^();

// Unused - Implemented for compatibility reason!
{attribute 'hide'}
METHOD OnBACnetRMObjectCOV
VAR_INPUT
	ePropID		: E_BACnetPropIdentifier;
END_VAR
END_METHOD

// Unused - Implemented for compatibility reason!
{attribute 'hide'}
METHOD OnBACnetRMObjectStateChanged
END_METHOD

METHOD FB_init : BOOL
VAR_INPUT
	bInitRetains : BOOL; // if TRUE, the retain variables are initialized (warm start / cold start)
	bInCopyCode : BOOL;  // if TRUE, the instance afterwards gets moved into the copy code (online change)
END_VAR
iOwner := THIS^;
END_METHOD

{attribute 'suppress_wrn_C0410'}
{attribute 'hide'}
PROPERTY LogMsg : REFERENCE TO FB_BA_LogMessage
GET
LogMsg REF= fbLogMsg;
END_GET
END_PROPERTY

END_FUNCTION_BLOCK

// POUs/Remote/Objects/Basic/[Internal]/FB_BACnetRM_BaseObject
FUNCTION_BLOCK FB_BACnetRM_BaseObject IMPLEMENTS I_BACnetRM_BaseObject
VAR_INPUT CONSTANT
	{region 'Fixed Parameters'}
		{attribute 'parameterCategory':='General'}
		{attribute 'no_copy'}
		Client : REFERENCE TO FB_BACnet_Client;
		{attribute 'parameterCategory':='General'}
		nObjectInstance : UDINT := BACnet_Globals.nBACnetInstId_Auto;	
		{attribute 'parameterCategory':='Communication'}
		eReadMode : E_BACnet_CommMode := E_BACnet_CommMode.eAuto;
	{endregion}
END_VAR
VAR_OUTPUT
	bReady					: BOOL;
END_VAR
VAR
	{region 'SubInit'}
		eObjectType			: E_BACnetObjType				:= 16#FFFF;
		{attribute 'hide'}
		iOwner				: I_BACnetRM_ObjectOwner;												// Owner of current Instance (Pointer to current instance per default)
	{endregion}
END_VAR
VAR
	{region 'General'}
		eErrorID			: E_BACnet_Error				:= E_BACnet_Error.eNoError;
			 
		tObjectID			: T_BACnet_ObjectIdentifier		:= 16#FFFFFFFF;
			 
		{attribute 'hide'}
		{attribute 'no_copy'}
		bInit				: BOOL;
	{endregion}
END_VAR

IF (NOT bReady) THEN
	IF (iOwner = 0) THEN
		eErrorID := E_BACnet_Error.eInvalidParameter;
		F_BA_LogMessage(ADSLOG_MSGTYPE_ERROR, 'O04', 'Owner of BACnet remote-object not defined!');
		
	ELSIF (__ISVALIDREF(Client)) THEN
		IF (NOT Client.bConnected) THEN		
			; // Wait for referred client to be conntected.
		ELSE
			IF NOT bInit THEN
				bInit := TRUE;
				OnObjectStateChanged();
				tObjectID := F_BACnet_GetObjId(eObjectType, nObjectInstance);		
				Client.UpdateRequests();
			ELSE
				IF Client.bReady THEN
					eErrorID := E_BACnet_Error.eNoError;
					bReady := TRUE;
				END_IF
			END_IF
		END_IF
	ELSE
		eErrorID := E_BACnet_Error.eInvalidClient;
		iOwner.LogMsg.Show(ADSLOG_MSGTYPE_ERROR, 'O17', 'Assigned client-reference is invalid!', FALSE);
	END_IF
ELSE
	IF NOT Client.bReady THEN
		bReady := FALSE;
	END_IF
END_IF

{attribute 'hide'}
METHOD OnCOV
VAR_INPUT
	ePropID		: E_BACnetPropIdentifier;
END_VAR
// Notify owner:
iOwner.OnBACnetRMObjectCOV(ePropID);
END_METHOD

{attribute 'hide'}
METHOD OnReqError
VAR_INPUT
	iRequest		: I_BACnetRM_BaseReq;
	stResult		: POINTER TO SendDataRequestResult;
	sLogCode		: STRING			:= '';
END_VAR
VAR_STAT
	// (BETA) ... Following symbols should be made non-static / thread safe!
	_sTemp			: STRING;
	fbMessage		: FB_BA_DecorMessage;
END_VAR
fbMessage.Reset();

IF (stResult = 0) THEN
	iOwner.LogMsg.Show(ADSLOG_MSGTYPE_ERROR, 'ORE04', 'Internal error in implementation of error-handling!', FALSE);
ELSE
	CASE (stResult^.errorType) OF
		E_BACnet_ErrorType.eError:
			IF (NOT F_BACnet_IsErrorClassValid(TO_INT(stResult^.errorClass))) THEN
				iOwner.LogMsg.Show1(ADSLOG_MSGTYPE_ERROR, 'ORE07', 'Received unknown error of invalid class "%d"!', F_DINT(stResult^.errorClass), FALSE);
			ELSIF (NOT F_BACnet_IsErrorCodeValid(TO_INT(stResult^.errorCode))) THEN
				iOwner.LogMsg.Show1(ADSLOG_MSGTYPE_ERROR, 'ORE09', 'Received unknown error of invalid code "%d"!', F_DINT(stResult^.errorCode), FALSE);
			ELSE
				fbMessage.FormatText1('Received error "%s"', F_STRINGEx(BACnet_Globals.aSpec_ErrorCode[stResult^.errorCode]));
				fbMessage.AddDecor1('Class: %s', F_STRINGEx(BACnet_Globals.aSpec_ErrorClass[stResult^.errorClass]));
			END_IF
			
		E_BACnet_ErrorType.eReject:
			IF (NOT F_BACnet_IsRejectReasonValid(TO_INT(stResult^.rejectCode))) THEN
				iOwner.LogMsg.Show1(ADSLOG_MSGTYPE_ERROR, 'ORE16', 'Received unknown rejection of invalid reason "%d"!', F_DINT(stResult^.rejectCode), FALSE);
			ELSE
				fbMessage.FormatText1('Received rejection "%s".', F_STRINGEx(BACnet_Globals.aSpec_RejectReason[stResult^.rejectCode]));
			END_IF
		
		E_BACnet_ErrorType.eAbort:
			IF (NOT F_BACnet_IsAbortReasonValid(TO_INT(stResult^.abortReason))) THEN
				iOwner.LogMsg.Show1(ADSLOG_MSGTYPE_ERROR, 'ORE23', 'Received unknown abort of invalid reason "%d"!', F_DINT(stResult^.abortReason), FALSE);
			ELSE
				fbMessage.FormatText1('Received abort "%s".', F_STRINGEx(BACnet_Globals.aSpec_AbortReason[stResult^.abortReason]));
			END_IF
		
	ELSE
		iOwner.LogMsg.Show1(ADSLOG_MSGTYPE_ERROR, 'ORE29', 'Invalid error of type "%d" received!', F_DINT(stResult^.errorType), FALSE);
	END_CASE
END_IF

IF (NOT fbMessage.IsEmpty) THEN
	// Add further information:
	IF (bReady) THEN
		_sTemp := F_BACnet_GetObjectIdString(tObjectID);
		fbMessage.AddDecor2('Remote Object: [%d]%s', F_UDINT(Client.nDeviceInstance), F_STRINGEx(_sTemp));
	END_IF
	CASE (stResult^.errorClass) OF
		E_BACnet_ErrorClass.eProperty:
			fbMessage.AddDecor1('Property: %d', F_INT(stResult^.propertyIdentifier));
//		E_BACnet_ErrorClass.xxx:
//			fbMessage.AddDecor1('Invoke ID: %d', F_UDINT(stResult^.invokeId));
//		E_BACnet_ErrorClass.xxx:
//			fbMessage.AddDecor1('Process ID: %d', F_UDINT(stResult^.processId));
	END_CASE
	
	// Build message:
	IF (fbMessage.Finish()) THEN
		iOwner.LogMsg.Show(ADSLOG_MSGTYPE_ERROR, sLogCode, fbMessage.sOutput, TRUE);
	END_IF
END_IF
END_METHOD

METHOD PROTECTED OnObjectStateChanged
// Notify owner:
iOwner.OnBACnetRMObjectStateChanged();
END_METHOD

PROPERTY Error : BOOL
GET
Error := (eErrorID <> E_BACnet_Error.eNoError);
END_GET
END_PROPERTY

PROPERTY ObjectID : T_BACnet_ObjectIdentifier
GET
ObjectID := tObjectID;
END_GET
END_PROPERTY

PROPERTY ObjectInstance : UDINT
GET
ObjectInstance := nObjectInstance;
END_GET
SET
PUBLIC 
VAR
END_VAR
nObjectInstance:=ObjectInstance;
tObjectID := F_BACnet_GetObjId(eObjectType, nObjectInstance);
END_SET
END_PROPERTY

PROPERTY ObjectType : E_BACnetObjType
GET
ObjectType := eObjectType;
END_GET
SET
PUBLIC 
VAR
END_VAR
eObjectType:=ObjectType;
tObjectID := F_BACnet_GetObjId(eObjectType, nObjectInstance);
END_SET
END_PROPERTY

PROPERTY ReadMode : E_BACnet_CommMode
GET
ReadMode:=eReadMode;
END_GET
SET
eReadMode:=ReadMode;
END_SET
END_PROPERTY

METHOD SyncProperty : BOOL
VAR_INPUT
	ePropID		: E_BACnetPropIdentifier;
	nSize		: UDINT;
	pData		: PVOID;
	eSyncMode	: E_BA_SyncModeRM;
END_VAR
VAR_STAT
	stRdEntry	: POINTER TO ST_BACnetRM_ReadEntry;
	stWrtEntry	: POINTER TO ST_BACnetRM_WriteEntry;
END_VAR
SyncProperty:=SyncPropertyReal(ePropID, nSize, pData, eSyncMode, 0.0);
END_METHOD

METHOD SyncPropertyEnable : BOOL
VAR_INPUT
	ePropID		: E_BACnetPropIdentifier;
	nSize		: UDINT;
	pData		: PVOID;
	pEnable		: POINTER TO BOOL := 0;
	eSyncMode	: E_BA_SyncModeRM;
END_VAR
VAR_STAT
	// (BETA) ... Following symbols should be made non-static / thread safe!
	stWrtEntry	: POINTER TO ST_BACnetRM_WriteEntry;
END_VAR
SyncPropertyEnable:=SyncPropertyPrioReal(ePropID, nSize, pData, pEnable, 0, E_BACnet_Priority.Last, eSyncMode, 0.0);
END_METHOD

METHOD SyncPropertyIdx : BOOL
VAR_INPUT
	ePropID		: E_BACnetPropIdentifier;
	nSize		: UDINT;
	pData		: PVOID;
	nIndex		: INT(0..2);
	eSyncMode	: E_BA_SyncModeRM;
END_VAR
VAR_STAT
	// (BETA) ... Following symbols should be made non-static / thread safe!
	stRdEntry	: POINTER TO ST_BACnetRM_ReadEntry;
	stWrtEntry	: POINTER TO ST_BACnetRM_WriteEntry;
END_VAR
IF (0 <= nIndex) AND_THEN (nIndex <= 2) THEN
	CASE (eSyncMode) OF
		E_BA_SyncModeRM.eRead:
			IF (SyncPropertyIdx := Client.AddReadEntry(THIS^, ePropID, E_BACnet_Priority.Invalid, stResult=>stRdEntry)) THEN
				stRdEntry^.nData := nSize;
				stRdEntry^.pData := pData;
				stRdEntry^.nIndex := TO_UDINT(nIndex);
			END_IF
		
		E_BA_SyncModeRM.eWrite:
			iOwner.LogMsg.Show1(ADSLOG_MSGTYPE_ERROR, 'SPI11', 'Unimplemented Sync-Mode "%d"!', F_INT(eSyncMode), TRUE);
		
	ELSE
		iOwner.LogMsg.Show1(ADSLOG_MSGTYPE_ERROR, 'SPI14', 'Invalid Sync-Mode "%d"!', F_INT(eSyncMode), TRUE);
	END_CASE
ELSE
	iOwner.LogMsg.Show1(ADSLOG_MSGTYPE_ERROR, 'SPI17', 'Invalid parameter "Index=%d"!', F_INT(nIndex), TRUE);
END_IF
END_METHOD

METHOD SyncPropertyPrio : BOOL
VAR_INPUT
	ePropID		: E_BACnetPropIdentifier;
	nSize		: UDINT;
	pData		: PVOID;
	pEnable		: POINTER TO BOOL := 0;
	pNull		: POINTER TO BOOL := 0;
	ePriority	: E_BACnet_Priority := E_BACnet_Priority.Last;
	eSyncMode	: E_BA_SyncModeRM;
END_VAR
VAR_STAT
	// (BETA) ... Following symbols should be made non-static / thread safe!
	stWrtEntry	: POINTER TO ST_BACnetRM_WriteEntry;
END_VAR
SyncPropertyPrio:=SyncPropertyPrioReal(ePropID, nSize, pData, pEnable, pNull, ePriority, eSyncMode, 0.0);
END_METHOD

METHOD SyncPropertyPrioReal : BOOL
VAR_INPUT
	ePropID			: E_BACnetPropIdentifier;
	nSize			: UDINT;
	pData			: PVOID;
	pEnable			: POINTER TO BOOL := 0;
	pNull			: POINTER TO BOOL := 0;
	ePriority		: E_BACnet_Priority := E_BACnet_Priority.Last;
	eSyncMode		: E_BA_SyncModeRM;
	fCOVIncrement	: REAL;
END_VAR
VAR_STAT
	// (BETA) ... Following symbols should be made non-static / thread safe!
	stWrtEntry	: POINTER TO ST_BACnetRM_WriteEntry;
END_VAR
CASE (eSyncMode) OF
	E_BA_SyncModeRM.eRead:
		iOwner.LogMsg.Show1(ADSLOG_MSGTYPE_ERROR, 'SPP03', 'Unimplemented Sync-Mode "%d"!', F_INT(eSyncMode), TRUE);
	
	E_BA_SyncModeRM.eWrite:
		IF (SyncPropertyPrioReal := Client.AddWriteEntry(THIS^, ePropID, ePriority, stResult=>stWrtEntry)) THEN
			stWrtEntry^.nData := nSize;
			stWrtEntry^.pData := pData;
			stWrtEntry^.pEnable := pEnable;
			stWrtEntry^.pNull := pNull;
			stWrtEntry^.nPriority := TO_UDINT(ePriority);
			stWrtEntry^.fCOVIncrement := fCOVIncrement;
		END_IF
	
ELSE
	iOwner.LogMsg.Show1(ADSLOG_MSGTYPE_ERROR, 'SPP09', 'Invalid Sync-Mode "%d"!', F_INT(eSyncMode), TRUE);
END_CASE
END_METHOD

METHOD SyncPropertyReal : BOOL
VAR_INPUT
	ePropID			: E_BACnetPropIdentifier;
	nSize			: UDINT;
	pData			: PVOID;
	eSyncMode		: E_BA_SyncModeRM;
	fCOVIncrement	: REAL;
END_VAR
VAR_STAT
	stRdEntry	: POINTER TO ST_BACnetRM_ReadEntry;
	stWrtEntry	: POINTER TO ST_BACnetRM_WriteEntry;
END_VAR
CASE (eSyncMode) OF
	E_BA_SyncModeRM.eRead:
		IF (SyncPropertyReal := Client.AddReadEntry(THIS^, ePropID, E_BACnet_Priority.Invalid, stResult=>stRdEntry)) THEN
			stRdEntry^.nData := nSize;
			stRdEntry^.pData := pData;
			stRdEntry^.fCOVIncrement := fCOVIncrement;
		END_IF
	
	E_BA_SyncModeRM.eWrite:
		IF (SyncPropertyReal := Client.AddWriteEntry(THIS^, ePropID, E_BACnet_Priority.Invalid, stResult=>stWrtEntry)) THEN
			stWrtEntry^.nData := nSize;
			stWrtEntry^.pData := pData;
			stWrtEntry^.fCOVIncrement := fCOVIncrement;
		END_IF
	
ELSE
	iOwner.LogMsg.Show1(ADSLOG_MSGTYPE_ERROR, 'SP09', 'Invalid Sync-Mode "%d"!', F_INT(eSyncMode), TRUE);
END_CASE
END_METHOD

END_FUNCTION_BLOCK

// POUs/Remote/FB_BACnet_Client
{attribute 'enable_dynamic_creation'}
FUNCTION_BLOCK FB_BACnet_Client IMPLEMENTS I_BACnetRM_Object
VAR_INPUT CONSTANT
	{region 'Fixed Parameters'}
		{attribute 'parameterCategory':='General'}
		{attribute 'no_copy'}
		Adapter	: REFERENCE TO FB_BACnet_Adapter := BACnet_Globals.DefaultAdapter;
		{attribute 'parameterCategory':='General'}
		nDeviceInstance : UDINT;
	{endregion}
END_VAR
VAR_INPUT CONSTANT PERSISTENT
	{region 'Variable Parameters'}
		{attribute 'parameterCategory':='Communication'}
		nMaxParallelRequests : UDINT := 1;
		{attribute 'parameterCategory':='Communication'}
		nRPMPropertiesPerRequest : UDINT := 80;
		{attribute 'parameterCategory':='Communication'}
		tCOVLifeTime : TIME := T#240S;	
		{attribute 'parameterCategory':='Communication'}
		eReadMode : E_BACnet_CommMode := E_BACnet_CommMode.eAuto;
		{attribute 'parameterCategory':='Communication'}
		tReadCycleTime : TIME := T#5S;
		{attribute 'parameterCategory':='Communication'}
		tWriteCycleTime : TIME := T#5S;
		{attribute 'parameterCategory':='Supported Services'}
		bSuppRpm  : BOOL;
		{attribute 'parameterCategory':='Supported Services'}
		bSuppCov  : BOOL;
		{attribute 'parameterCategory':='Supported Services'}
		bSuppCovP : BOOL;
	{endregion}
END_VAR
VAR_OUTPUT
	bReady					: BOOL;
	eErrorID				: E_BACnet_Error;
	nAdsPort 				: UINT;
	bConnected  			: BOOL;
END_VAR
VAR
	{region 'General'}
		tObjectID			: T_BACnet_ObjectIdentifier		:= 16#FFFFFFFF;
	{endregion}
END_VAR
VAR
	{region 'General'}
		eState				: E_BACnetRM_ClientState;	
		stSupportedServices	: ST_BACnet_ServicesSupportedBits;
		nMaxApduSize 		: UDINT;
	{endregion}
	{region 'Request Lists'}
		{region 'Read'}
			{attribute 'hide'}
			stReadList 		: POINTER TO ST_BACnetRM_ReadEntry;
			{attribute 'hide'}
			nReadList		: UDINT := 0;
			{attribute 'hide'}
			nReadMax		: UDINT := 0;
		{endregion}
		{region 'Write'}
			{attribute 'hide'}
			stWriteList		: POINTER TO ST_BACnetRM_WriteEntry;
			{attribute 'hide'}
			nWriteList		: UDINT := 0;
			{attribute 'hide'}
			nWriteMax		: UDINT := 0;	
		{endregion}
	{endregion}
	{region 'Request Fifo'}
		{region 'Cyclic'}
			{attribute 'hide'}
			stReqList		: POINTER TO ST_BACnetRM_ReqPtr := 0;
			{attribute 'hide'}
			nReqList		: UDINT := 0;
			{attribute 'hide'}
			nCurReq			: UDINT := 0;
		{endregion}
		{region 'Acyclic / Dynamic'}
			{attribute 'hide'}
			fbReadFifo		: FB_BACnetRM_ReqFifo := (Client := THIS^);
			{attribute 'hide'}
			fbWriteFifo		: FB_BACnetRM_ReqFifo := (Client := THIS^);
		{endregion}
				  
		nOpenReq			: UDINT := 0;
		{attribute 'hide'}
		bUpdateReqs			: BOOL;
	{endregion}
		 
	{region 'Internal'}
		{attribute 'hide'}
		iServer				: ITcIoBACnetPlcServer;
		{attribute 'hide'}
		iClient				: ITcIoBACnetPlcClient;
		{attribute 'hide'}
		iDevice				: ITcIoBACnetPlcDevice;
		{attribute 'hide'}
		_bCreated			: BOOL;
			 
		{attribute 'hide'}
		fbRead				: FB_BACnetRM_ReadProperty := (Client:=THIS^);
		{attribute 'hide'}
		_ClientStatus		: WORD;
		{attribute 'hide'}
		_ClientControl		: WORD;
		{attribute 'hide'}
		_tReInitTime		: TIME;
		{attribute 'hide'}
		_tCycleStartTime	: TIME;
		diagCycleDuration 	: TIME;
	{endregion}
END_VAR
VAR_STAT
	// (BETA) ... Following symbols should be made non-static / thread safe!
	{region 'Temporary'}
		_n					: UDINT;
		_nRpmTreshold		: UDINT;
	{endregion}
END_VAR

IF (__ISVALIDREF(Adapter)) THEN
	Adapter();
	
	IF (iDevice = 0) THEN
		iDevice := Adapter.Device;
	END_IF
END_IF

IF iClient = 0 THEN
	IF iDevice <> 0 THEN
		IF S_OK <> iDevice.GetClientById(nDeviceInstance, ADR(iServer)) THEN
			IF NOT _bCreated THEN
				IF S_OK = iDevice.CreateClient(nDeviceInstance) THEN
					_bCreated := TRUE;
				END_IF
			END_IF			
		ELSE
			iServer.GetAdsPort(ADR(nAdsPort));
			IF S_OK <> iServer.TcQueryInterface(TC_GLOBAL_IID_LIST.IID_ITcIoBACnetPlcClient, ADR(iClient)) THEN
				eErrorID := E_BACnet_Error.eInvalidClient;
			END_IF
		END_IF
	END_IF
END_IF

IF iClient <> 0 THEN
	iServer.UpdateDeviceStatus(ADR(_ClientControl), ADR(_ClientStatus));	
	IF Adapter.bEthernetLink THEN
		bConnected := NOT (SHR((_ClientStatus AND 16#FF00), 8) < 4);
	ELSE
		bConnected := FALSE;
	END_IF
	CASE eState OF
		E_BACnetRM_ClientState.eInit:
			IF bConnected THEN
				tObjectID := F_BACnet_GetObjId(ObjectType, nDeviceInstance);
				IF stSupportedServices.bSuppReadProperty THEN
					State:=E_BACnetRM_ClientState.eCalcAuto;
				ELSE
					State:=E_BACnetRM_ClientState.eReadSupportedServices;
				END_IF
			END_IF
		E_BACnetRM_ClientState.eReadSupportedServices:
			IF fbRead.bReady OR fbRead.bError THEN
				IF fbRead.bError THEN
					State:=E_BACnetRM_ClientState.eError;
				ELSE
					State:=E_BACnetRM_ClientState.eReadApduSize;
				END_IF
				fbRead(bExecute:=FALSE);
			ELSIF NOT fbRead.bBusy THEN
				fbRead(iObject:=THIS^, ePropID:=E_BACnetPropIdentifier.PropProtocolServicesSupported, nData:=SIZEOF(stSupportedServices), pData:=ADR(stSupportedServices), bExecute:=TRUE);
			END_IF
			fbReadFifo.ProcessReadFifo();
		E_BACnetRM_ClientState.eReadApduSize:
			IF fbRead.bReady OR fbRead.bError THEN
				IF fbRead.bError THEN
					State:=E_BACnetRM_ClientState.eError;
				ELSE
					State:=E_BACnetRM_ClientState.eCalcAuto;
				END_IF
				fbRead(bExecute:=FALSE);
			ELSIF NOT fbRead.bBusy THEN
				fbRead(iObject:=THIS^, ePropID:=E_BACnetPropIdentifier.PropMaxApduLengthAccepted, nData:=SIZEOF(nMaxApduSize), pData:=ADR(nMaxApduSize), bExecute:=TRUE);
			END_IF
			fbReadFifo.ProcessReadFifo();				
		E_BACnetRM_ClientState.eCalcAuto:
			IF nReadList>0 OR nWriteList>0 THEN
				IF eReadMode = E_BACnet_CommMode.eAuto THEN
					IF nMaxApduSize <= 480 THEN
						// [MS/TP Device]
						// > starting at 5 requests use RPM instead COV:
						_nRpmTreshold := 5;
						IF nMaxApduSize <= 206 THEN
							// For very small devices put only 10 properties into 1 request (prevent segmentation)
							nRPMPropertiesPerRequest := 10;
						ELSE
							nRPMPropertiesPerRequest := 20; 
						END_IF
					ELSE
						// [IP Device]
						// > Use more parallel requests
						nMaxParallelRequests := 50;
						_nRpmTreshold := 300;
					END_IF
					
					IF nReadList > _nRpmTreshold AND stSupportedServices.bSuppReadPropertyMultiple THEN
						eReadMode := E_BACnet_CommMode.eRpm;
					ELSIF stSupportedServices.bSuppSubscribeCOV THEN
						eReadMode := E_BACnet_CommMode.eCov;
					ELSIF stSupportedServices.bSuppReadPropertyMultiple THEN
						eReadMode := E_BACnet_CommMode.eRpm;
					ELSE
						eReadMode := E_BACnet_CommMode.eRp;
					END_IF
					bSuppRpm  := stSupportedServices.bSuppReadPropertyMultiple;
					bSuppCov  := stSupportedServices.bSuppSubscribeCov;
					bSuppCovP := stSupportedServices.bSuppSubscribeCOVProperty; 
				END_IF
				State:=E_BACnetRM_ClientState.eCreateRequests;
			ELSE
				State:=E_BACnetRM_ClientState.eCycle;
			END_IF
			State:=E_BACnetRM_ClientState.eCreateRequests;
		E_BACnetRM_ClientState.eCreateRequests:
			IF eReadMode = E_BACnet_CommMode.eAuto OR eReadMode = E_BACnet_CommMode.eRpm THEN
				fbReadFifo.bRpm:=stSupportedServices.bSuppReadPropertyMultiple;
			END_IF
			IF CreateReqList() THEN
				bUpdateReqs := FALSE;
				State:=E_BACnetRM_ClientState.eCycle;
			END_IF
		E_BACnetRM_ClientState.eCycle:
			IF bUpdateReqs THEN
				State:=E_BACnetRM_ClientState.eReInit;
				bUpdateReqs := FALSE;
				bReady:=FALSE;
			ELSE
				bReady:=TRUE;
				
				// Work on acyclic / dynamic requests:
				fbReadFifo.ProcessReadFifo();
				fbWriteFifo.ProcessWriteFifo();
				
				// Work on cyclic requests:
				IF stReqList <> 0 THEN
					_n := 0;
					WHILE nOpenReq < nMaxParallelRequests AND _n<nReqList DO								
						IF stReqList[nCurReq].pPtr <> 0 AND_THEN stReqList[nCurReq].fbBase^.IsReady() THEN
							IF stReqList[nCurReq].fbBase^.Send() THEN
								nOpenReq:=nOpenReq+1;
								IF nCurReq = 0 THEN
									IF _tCycleStartTime <> T#0S THEN
										diagCycleDuration:= TIME() - _tCycleStartTime;
									END_IF
									_tCycleStartTime := TIME();
								END_IF
							END_IF
						END_IF
						_n:=_n+1;
						nCurReq:=(nCurReq+1) MOD nReqList;
					END_WHILE
				END_IF
			END_IF
			IF NOT bConnected THEN
				State:=E_BACnetRM_ClientState.eReInit;
			END_IF
		E_BACnetRM_ClientState.eReInit:
			DeleteReqList();
			State:=E_BACnetRM_ClientState.eInit;
		E_BACnetRM_ClientState.eError:
			IF ((TIME()-_tReInitTime) > T#5S) THEN
				State:=E_BACnetRM_ClientState.eReInit;
			END_IF
	END_CASE
END_IF

{attribute 'hide'}
METHOD OnCOV
VAR_INPUT
	ePropID		: E_BACnetPropIdentifier;
END_VAR
END_METHOD

{attribute 'hide'}
METHOD OnReqError
VAR_INPUT
	iRequest		: I_BACnetRM_BaseReq;
	stResult		: POINTER TO SendDataRequestResult;
	sLogCode		: STRING			:= '';
END_VAR
VAR
	nLogType		: DWORD;
END_VAR
END_METHOD

METHOD INTERNAL OnRequestComplete
IF nOpenReq > 0 THEN
	nOpenReq:=nOpenReq-1;
END_IF
END_METHOD

METHOD INTERNAL AddReadEntry : BOOL
VAR_INPUT
	iObject 	: I_BACnetRM_BaseObject;
	ePropID 	: E_BACnetPropIdentifier;
	ePriority	: E_BACnet_Priority := E_BACnet_Priority.Invalid;
END_VAR
VAR_OUTPUT
	stResult	: POINTER TO ST_BACnetRM_ReadEntry;
END_VAR
VAR
	nTmp		: UDINT;
	nTmpSize	: UDINT;
	pTmp		: PVOID;
END_VAR
// Search for existing entry:
FOR nTmp := nReadList TO 1 BY -1 DO
	stResult := ADR(stReadList[nTmp-1]);
	IF (stResult^.iObject = iObject) AND_THEN (stResult^.ePropID = ePropID) THEN
		F_BA_LogMessage1(ADSLOG_MSGTYPE_ERROR, 'ARE05', 'Failed to initialize duplicate RemoteRead-Entry for Property "%d"!', F_INT(ePropID));
		RETURN;
	END_IF
END_FOR

IF (nReadList+1 >= nReadMax) THEN
	// Append list:
	nTmp := nReadMax+10;
	nTmpSize := nTmp*SIZEOF(ST_BACnetRM_ReadEntry);
	pTmp := __NEW(BYTE,nTmpSize);
	IF pTmp = 0 THEN
		RETURN;
	END_IF
	IF stReadList <> 0 THEN
		MEMCPY(pTmp, stReadList, nReadMax*SIZEOF(ST_BACnetRM_ReadEntry));
		__DELETE(stReadList);
	END_IF
	stReadList:=pTmp;
	nReadMax:=nTmp;
END_IF

// Create new entry:
stResult := ADR(stReadList[nReadList]);
nReadList := (nReadList+1);

// Initialize entry:
MEMSET(stResult, 0, SIZEOF(ST_BACnetRM_ReadEntry));
stResult^.iObject := iObject;
stResult^.ePropID := ePropID;
stResult^.nIndex := 16#FFFFFFFF;

AddReadEntry:=TRUE;
END_METHOD

METHOD INTERNAL AddWriteEntry : BOOL
VAR_INPUT
	iObject 	: I_BACnetRM_BaseObject;
	ePropID 	: E_BACnetPropIdentifier;
	ePriority	: E_BACnet_Priority := E_BACnet_Priority.Invalid;
END_VAR
VAR_OUTPUT
	stResult	: POINTER TO ST_BACnetRM_WriteEntry;
END_VAR
VAR
	nTmp		: UDINT;
	nTmpSize	: UDINT;
	pTmp		: PVOID;
END_VAR
// Search for existing entry:
FOR nTmp := nWriteList TO 1 BY -1 DO
	stResult := ADR(stWriteList[nTmp-1]);
	IF (stResult^.iObject = iObject) AND_THEN (stResult^.ePropID = ePropID) THEN
		IF (ePropID = E_BACnetPropIdentifier.PropPresentValue) AND_THEN (stResult^.nPriority <> TO_UDINT(ePriority)) THEN
			; // Allow requests on different priorities.
		ELSE
			F_BA_LogMessage1(ADSLOG_MSGTYPE_ERROR, 'AWE05', 'Failed to initialize duplicate RemoteWrite-Entry for Property "%d"!', F_INT(ePropID));
			RETURN;
		END_IF
	END_IF
END_FOR

IF (nWriteList+1 >= nWriteMax) THEN
	// Append list:
	nTmp := nWriteMax+10;
	nTmpSize := nTmp*SIZEOF(ST_BACnetRM_WriteEntry);
	pTmp := __NEW(BYTE,nTmpSize);
	IF pTmp = 0 THEN
		RETURN;
	END_IF
	IF stWriteList <> 0 THEN
		MEMCPY(pTmp, stWriteList, nWriteMax*SIZEOF(ST_BACnetRM_WriteEntry));
		__DELETE(stWriteList);
	END_IF
	stWriteList:=pTmp;
	nWriteMax:=nTmp;
END_IF

// Create new entry:
stResult := ADR(stWriteList[nWriteList]);
nWriteList := (nWriteList+1);

// Initialize entry:
MEMSET(stResult, 0, SIZEOF(ST_BACnetRM_WriteEntry));
stResult^.iObject := iObject;
stResult^.ePropID := ePropID;
stResult^.fCOVIncrement := 0.0;

AddWriteEntry := TRUE;
END_METHOD

METHOD INTERNAL AddFifoReadReq : BOOL
VAR_INPUT
	pReq : POINTER TO FB_BACnetRM_ReadProperty;
END_VAR
VAR
	entry : ST_BACnetRM_FifoEntry;
END_VAR
entry.fbRead:=pReq;
AddFifoReadReq:=fbReadFifo.AddFifoReq(entry);
END_METHOD

METHOD INTERNAL AddFifoWriteReq : BOOL
VAR_INPUT
	pReq : POINTER TO FB_BACnetRM_WriteProperty;
END_VAR
VAR
	entry : ST_BACnetRM_FifoEntry;
END_VAR
entry.fbWrite:=pReq;
AddFifoWriteReq:=fbWriteFifo.AddFifoReq(entry);
END_METHOD

{attribute 'hide'}
METHOD UpdateRequests 
VAR_INPUT
END_VAR
bUpdateReqs:=TRUE;
bReady:=FALSE;
END_METHOD

METHOD PRIVATE CreateReadReq : I_BACnetRM_BaseReq
VAR_INPUT
	eReadMode : E_BACnet_CommMode;
	stEntry : ST_BACnetRM_ReadEntry;
END_VAR
VAR
	stPtr : ST_BACnetRM_ReqPtr;
END_VAR
CASE eReadMode OF
	E_BACnet_CommMode.eCov:
		stPtr.fbCov:=__NEW(FB_BACnetRM_ReqCov);
		IF stPtr.fbCov <> 0 THEN
			stPtr.fbCov^(Client:=THIS^,iObject:=stEntry.iObject,  ePropID:=stEntry.ePropID, tLifetime:=tCOVLifeTime, pData:=stEntry.pData, nData:=stEntry.nData);
			stPtr.fbCov^.InitTimer();
		END_IF
		CreateReadReq:=stPtr.iReq;
		RETURN;
	E_BACnet_CommMode.eCovC:
		stPtr.fbCov:=__NEW(FB_BACnetRM_ReqCov);
		IF stPtr.fbCov <> 0 THEN
			stPtr.fbCov^(Client:=THIS^,iObject:=stEntry.iObject, bConfirmed:=TRUE, ePropID:=stEntry.ePropID, tLifetime:=tCOVLifeTime, pData:=stEntry.pData, nData:=stEntry.nData);
			stPtr.fbCov^.InitTimer();
		END_IF
		CreateReadReq:=stPtr.iReq;
		RETURN;
	E_BACnet_CommMode.eCovU:
		stPtr.fbCov:=__NEW(FB_BACnetRM_ReqCov);
		IF stPtr.fbCov <> 0 THEN
			stPtr.fbCov^(Client:=THIS^,iObject:=stEntry.iObject, bUnsubscribed:=TRUE, ePropID:=stEntry.ePropID, tLifetime:=tCOVLifeTime, pData:=stEntry.pData, nData:=stEntry.nData);
			stPtr.fbCov^.InitTimer();
		END_IF
		CreateReadReq:=stPtr.iReq;
		RETURN;
	E_BACnet_CommMode.eRp:
		stPtr.fbRead:=__NEW(FB_BACnetRM_ReqRead);
		IF stPtr.fbRead <> 0 THEN
			stPtr.fbRead^(Client:=THIS^,iObject:=stEntry.iObject, tCycleTime:=tReadCycleTime, ePropID:=stEntry.ePropID, pData:=stEntry.pData, nData:=stEntry.nData);
			stPtr.fbRead^.InitTimer();
		END_IF
		CreateReadReq:=stPtr.iReq;
		RETURN;
	E_BACnet_CommMode.eRpm:
		stPtr.fbRpm:=__NEW(FB_BACnetRM_ReqRpm);
		IF stPtr.fbRpm <> 0 THEN
			stPtr.fbRpm^(Client:=THIS^,iObject:=stEntry.iObject, tCycleTime:=tReadCycleTime);
			stPtr.fbRpm^.InitTimer();
		END_IF
		CreateReadReq:=stPtr.iReq;
		RETURN;
END_CASE
END_METHOD

METHOD PRIVATE CreateReqList : BOOL
VAR_INPUT
END_VAR
VAR
	i : UDINT;
	n : UDINT;
	nRpmEntries : UDINT;
	nReqs : UDINT;
	stPtr : ST_BACnetRM_ReqPtr;
	nReqsLeft : UDINT;
	pCurRpmReq : POINTER TO FB_BACnetRM_ReqRpm;
	bOptimizeCov : BOOL;
	nSize : UDINT;
END_VAR
DeleteReqList();

IF nReadList = 0 THEN
	CreateReqList:=TRUE;
	RETURN;
END_IF

// Calculate effective access mode and count RPM entries
FOR i:=0 TO nReadList-1 DO
	IF stReadList[i].iObject.ReadMode = E_BACnet_CommMode.eAuto THEN
		stReadList[i].eReadMode := eReadMode;
	ELSE
		stReadList[i].eReadMode := stReadList[i].iObject.ReadMode;
	END_IF
	IF F_IsCovReadMode(stReadList[i].eReadMode) THEN
		IF NOT bSuppCovP THEN
			IF NOT F_IsCovProperty(stReadList[i].iObject.ObjectType, stReadList[i].ePropID) THEN
				// ggf. error message if stReadList[i].fCOVIncrement <> 0.0
				IF bSuppRpm THEN
					stReadList[i].eReadMode := E_BACnet_CommMode.eRpm;
				ELSE
					stReadList[i].eReadMode := E_BACnet_CommMode.eRp;
				END_IF
			END_IF
		END_IF
		IF NOT bSuppCov THEN
			// ggf. error message that COV is configured but not available
			IF bSuppRpm THEN
				stReadList[i].eReadMode := E_BACnet_CommMode.eRpm;
			ELSE
				stReadList[i].eReadMode := E_BACnet_CommMode.eRp;
			END_IF
		END_IF
	END_IF
	IF stReadList[i].eReadMode = E_BACnet_CommMode.eRpm THEN
		nRpmEntries:=nRpmEntries+1;
	END_IF
END_FOR

// Calculate RPM request count
IF nRpmEntries > 0 THEN
	nReqs:=((nRpmEntries+nRPMPropertiesPerRequest-1)/nRPMPropertiesPerRequest);
END_IF

// Add single read requests + write repuests
nReqs := nReqs + (nReadList-nRpmEntries) + nWriteList;

stReqList:=__NEW(POINTER TO ST_BACnetRM_ReqPtr, nReqs);

IF stReqList = 0 THEN
	RETURN;
END_IF

FOR i:=0 TO nReadList-1 DO
	IF stReadList[i].eReadMode = E_BACnet_CommMode.eRpm THEN
		IF pCurRpmReq = 0 OR_ELSE pCurRpmReq^.nEntries = nRPMPropertiesPerRequest THEN
			stPtr.fbRpm:=__NEW(FB_BACnetRM_ReqRpm);
			IF stPtr.fbRpm = 0 THEN
				RETURN;
			END_IF
			nSize:=nRPMPropertiesPerRequest*SIZEOF(ST_BACnetRM_ReadEntry);
			stPtr.fbRpm^.pEntries:=__NEW(BYTE,nSize);
			IF stPtr.fbRpm^.pEntries = 0 THEN
				RETURN;
			END_IF
			IF pCurRpmReq <> 0 THEN
				pCurRpmReq^.InitTimer();
		 		pCurRpmReq^.UpdateRequest();		
			END_IF
			stPtr.fbRpm^.bFreeEntries:=TRUE;
			pCurRpmReq:=stPtr.fbRpm; 
			stPtr.fbRpm^(Client:=THIS^, iObject:=stReadList[i].iObject, tCycleTime:=tReadCycleTime);
			stReqList[nReqList]:=stPtr;		
	 		nReqList:=nReqList+1;
		END_IF 
		pCurRpmReq^.pEntries[pCurRpmReq^.nEntries]:=stReadList[i];
 		pCurRpmReq^.nEntries := pCurRpmReq^.nEntries + 1;	
	ELSE	
		stReqList[nReqList].iReq := CreateReadReq(stReadList[i].eReadMode, stReadList[i]);
		IF stReqList[nReqList].pPtr = 0 THEN
			RETURN;
		END_IF
		IF F_IsCovReadMode(stReadList[i].eReadMode) THEN
			bOptimizeCov := TRUE;
		END_IF
		nReqList:=nReqList+1;
	END_IF
END_FOR

IF pCurRpmReq <> 0 THEN
	stPtr.fbRpm^.InitTimer();
	stPtr.fbRpm^.UpdateRequest();
END_IF

IF bOptimizeCov THEN
	OptimizeCOV();
END_IF

IF (nWriteList > 0) THEN
	FOR i:=0 TO nWriteList-1 DO
		stReqList[nReqList].fbWrite := __NEW(FB_BACnetRM_ReqWrite);
		IF stReqList[nReqList].pPtr = 0 THEN
			RETURN;
		END_IF	
		stReqList[nReqList].fbWrite^(Client:=THIS^, iObject:=stWriteList[i].iObject, ePropID:=stWriteList[i].ePropID, tCycleTime:=tWriteCycleTime, pData:=stWriteList[i].pData, nData:=stWriteList[i].nData, pEnable:=stWriteList[i].pEnable, pNull:=stWriteList[i].pNull, fCOVIncrement:=stWriteList[i].fCOVIncrement, ePriority:=TO_INT(stWriteList[i].nPriority));
		stReqList[nReqList].fbWrite^.InitTimer();
		nReqList:=nReqList+1;
	END_FOR
END_IF

nCurReq := 0;
nOpenReq := 0;
CreateReqList:=TRUE;
END_METHOD

METHOD PRIVATE DeleteReqList
VAR_INPUT
END_VAR
VAR
	i : UDINT;
END_VAR
IF nReqList > 0 AND stReqList <> 0 THEN
	FOR i:=0 TO nReqList-1 DO
		IF stReqList[i].nByte <> 0 THEN
			CASE stReqList[i].iReq.GetRequestType() OF
				E_BACnetRM_RequestType.eRead:__DELETE(stReqList[i].fbRead);
				E_BACnetRM_RequestType.eReadPropertyMultiple:__DELETE(stReqList[i].fbRpm); 
				E_BACnetRM_RequestType.eWrite:__DELETE(stReqList[i].fbWrite);
				E_BACnetRM_RequestType.eWritePropertyMultiple:__DELETE(stReqList[i].fbWpm);
				E_BACnetRM_RequestType.eCOV_C:__DELETE(stReqList[i].fbCov);
				E_BACnetRM_RequestType.eCOV:__DELETE(stReqList[i].fbCov);
				E_BACnetRM_RequestType.eCOV_U:__DELETE(stReqList[i].fbCov);
			END_CASE
		END_IF
	END_FOR
	__DELETE(stReqList);
	stReqList:=0;
	nReqList:=0;
END_IF
END_METHOD

